C05450=1081.864,342.520,-93.492,176.172,26.985,154.564
C05451=1081.871,342.768,-93.526,176.175,26.990,154.565
C05452=1081.876,343.015,-93.561,176.178,26.994,154.566
C05453=1081.883,343.263,-93.595,176.181,27.000,154.567
C05454=1081.892,343.670,-93.651,176.186,27.008,154.568
C05455=1081.902,344.077,-93.708,176.192,27.016,154.570
C05456=1081.912,344.484,-93.765,176.197,27.024,154.571
C05457=1081.922,344.891,-93.822,176.202,27.033,154.572
C05458=1081.928,345.139,-93.856,176.205,27.038,154.573
C05459=1081.934,345.386,-93.892,176.208,27.043,154.574
C05460=1081.940,345.634,-93.926,176.212,27.048,154.575
C05461=1081.946,345.881,-93.960,176.215,27.053,154.576
C05462=1081.952,346.129,-93.996,176.218,27.058,154.577
C05463=1081.958,346.376,-94.030,176.221,27.063,154.577
C05464=1081.964,346.624,-94.066,176.224,27.068,154.578
C05465=1081.970,346.871,-94.100,176.228,27.074,154.579
C05466=1081.976,347.119,-94.135,176.231,27.078,154.580
C05467=1081.982,347.366,-94.169,176.234,27.084,154.581
C05468=1081.988,347.614,-94.204,176.237,27.088,154.582
C05469=1081.994,347.861,-94.239,176.241,27.094,154.582
C05470=1082.000,348.109,-94.274,176.244,27.099,154.583
C05471=1082.006,348.356,-94.309,176.247,27.104,154.584
C05472=1082.012,348.603,-94.344,176.251,27.110,154.585
C05473=1082.017,348.851,-94.379,176.254,27.115,154.586
C05474=1082.024,349.098,-94.414,176.256,27.120,154.587
C05475=1082.030,349.347,-94.449,176.259,27.125,154.588
C05476=1082.036,349.593,-94.484,176.263,27.130,154.589
C05477=1082.042,349.841,-94.519,176.266,27.136,154.589
C05478=1082.048,350.088,-94.553,176.269,27.141,154.590
C05479=1082.054,350.336,-94.589,176.272,27.146,154.591
C05480=1082.061,350.583,-94.624,176.276,27.152,154.592
C05481=1082.066,350.831,-94.659,176.279,27.156,154.593
C05482=1082.073,351.078,-94.694,176.282,27.162,154.594
C05483=1082.078,351.325,-94.729,176.286,27.167,154.595
C05484=1082.084,351.573,-94.765,176.289,27.172,154.596
C05485=1082.091,351.821,-94.800,176.292,27.178,154.597
C05486=1082.096,352.068,-94.835,176.296,27.183,154.598
C05487=1082.103,352.315,-94.870,176.299,27.188,154.598
C05488=1082.109,352.563,-94.906,176.302,27.194,154.599
C05489=1082.115,352.811,-94.942,176.305,27.199,154.600
C05490=1082.121,353.058,-94.976,176.308,27.204,154.601
C05491=1082.127,353.306,-95.011,176.311,27.210,154.602
C05492=1082.133,353.553,-95.047,176.315,27.215,154.603
C05493=1082.139,353.800,-95.082,176.318,27.220,154.604
C05494=1082.145,354.048,-95.118,176.321,27.226,154.605
C05495=1082.151,354.295,-95.153,176.325,27.232,154.606
C05496=1082.156,354.542,-95.189,176.328,27.237,154.607
C05497=1082.163,354.790,-95.224,176.331,27.242,154.608
C05498=1082.169,355.037,-95.260,176.335,27.248,154.609
C05499=1082.175,355.284,-95.295,176.338,27.253,154.610
C05500=1082.181,355.532,-95.331,176.340,27.258,154.611
C05501=1082.187,355.780,-95.366,176.344,27.264,154.611
C05502=1082.194,356.026,-95.402,176.347,27.270,154.612
C05503=1082.199,356.273,-95.438,176.350,27.275,154.613
C05504=1082.205,356.521,-95.473,176.354,27.280,154.614
C05505=1082.211,356.769,-95.509,176.357,27.286,154.615
C05506=1082.222,357.179,-95.568,176.362,27.295,154.617
C05507=1082.232,357.589,-95.627,176.368,27.304,154.618
C05508=1082.242,357.998,-95.687,176.374,27.313,154.620
C05509=1082.251,358.408,-95.746,176.379,27.322,154.622
C05510=1082.258,358.656,-95.781,176.383,27.328,154.623
C05511=1082.265,358.903,-95.818,176.386,27.334,154.624
C05512=1082.271,359.150,-95.853,176.388,27.339,154.625
C05513=1082.277,359.398,-95.889,176.392,27.345,154.625
C05514=1082.283,359.645,-95.925,176.395,27.351,154.626
C05515=1082.288,359.892,-95.961,176.399,27.357,154.628
C05516=1082.295,360.139,-95.997,176.402,27.362,154.628
C05517=1082.301,360.387,-96.033,176.405,27.367,154.629
C05518=1082.307,360.635,-96.069,176.409,27.373,154.630
C05519=1082.313,360.882,-96.105,176.412,27.379,154.632
C05520=1082.319,361.129,-96.141,176.416,27.385,154.632
C05521=1082.325,361.376,-96.177,176.418,27.390,154.633
C05522=1082.332,361.624,-96.213,176.421,27.396,154.635
C05523=1082.337,361.870,-96.249,176.425,27.402,154.636
C05524=1082.344,362.117,-96.286,176.428,27.408,154.637
C05525=1082.350,362.365,-96.321,176.432,27.413,154.637
C05526=1082.356,362.612,-96.358,176.435,27.419,154.639
C05527=1082.362,362.860,-96.394,176.439,27.425,154.640
C05528=1082.368,363.107,-96.431,176.442,27.431,154.641
C05529=1082.374,363.354,-96.467,176.445,27.437,154.642
C05530=1082.380,363.602,-96.503,176.448,27.442,154.643
C05531=1082.386,363.849,-96.539,176.452,27.448,154.644
C05532=1082.393,364.096,-96.576,176.455,27.454,154.645
C05533=1082.399,364.343,-96.612,176.458,27.460,154.646
C05534=1082.405,364.591,-96.648,176.462,27.466,154.647
C05535=1082.411,364.838,-96.684,176.465,27.471,154.648
C05536=1082.417,365.085,-96.721,176.468,27.477,154.649
C05537=1082.423,365.332,-96.758,176.471,27.483,154.650
C05538=1082.430,365.579,-96.794,176.475,27.489,154.651
C05539=1082.436,365.826,-96.831,176.478,27.495,154.652
C05540=1082.442,366.074,-96.868,176.482,27.501,154.653
C05541=1082.448,366.321,-96.903,176.485,27.507,154.654
C05542=1082.454,366.568,-96.940,176.489,27.513,154.655
C05543=1082.459,366.816,-96.977,176.491,27.519,154.656
C05544=1082.466,367.063,-97.013,176.495,27.525,154.658
C05545=1082.472,367.310,-97.050,176.498,27.531,154.659
C05546=1082.478,367.557,-97.087,176.502,27.538,154.660
C05547=1082.484,367.804,-97.123,176.505,27.543,154.661
C05548=1082.490,368.052,-97.160,176.509,27.550,154.662
C05549=1082.496,368.298,-97.197,176.511,27.555,154.663
C05550=1082.503,368.545,-97.234,176.515,27.562,154.664
C05551=1082.509,368.793,-97.271,176.518,27.567,154.665
C05552=1082.515,369.040,-97.308,176.522,27.574,154.666
C05553=1082.521,369.288,-97.345,176.526,27.580,154.667
C05554=1082.527,369.535,-97.381,176.529,27.586,154.669
C05555=1082.533,369.782,-97.418,176.532,27.592,154.670
C05556=1082.539,370.029,-97.455,176.535,27.598,154.671
C05557=1082.546,370.276,-97.492,176.539,27.605,154.672
C05558=1082.552,370.489,-97.524,176.542,27.610,154.673
C05559=1082.556,370.701,-97.556,176.545,27.615,154.674
C05560=1082.562,370.915,-97.588,176.547,27.620,154.675
C05561=1082.567,371.128,-97.619,176.550,27.625,154.676
C05562=1082.572,371.340,-97.651,176.553,27.631,154.677
C05563=1082.578,371.554,-97.684,176.556,27.636,154.678
C05564=1082.583,371.766,-97.715,176.559,27.642,154.679
C05565=1082.589,371.979,-97.747,176.562,27.647,154.680
C05566=1082.594,372.227,-97.784,176.566,27.653,154.681
C05567=1082.601,372.474,-97.821,176.569,27.660,154.682
C05568=1082.607,372.721,-97.859,176.572,27.666,154.683
C05569=1082.614,372.968,-97.895,176.576,27.672,154.684
C05570=1082.619,373.215,-97.933,176.579,27.679,154.685
C05571=1082.626,373.462,-97.970,176.583,27.685,154.687
C05572=1082.632,373.709,-98.008,176.586,27.691,154.688
C05573=1082.639,373.956,-98.044,176.590,27.698,154.689
C05574=1082.645,374.203,-98.082,176.593,27.704,154.690
C05575=1082.650,374.450,-98.119,176.596,27.710,154.691
C05576=1082.657,374.698,-98.156,176.600,27.717,154.692
C05577=1082.663,374.944,-98.194,176.603,27.723,154.694
C05578=1082.669,375.192,-98.231,176.607,27.730,154.695
C05579=1082.675,375.438,-98.269,176.610,27.736,154.696
C05580=1082.682,375.686,-98.307,176.613,27.743,154.697
C05581=1082.688,375.933,-98.344,176.617,27.749,154.698
C05582=1082.694,376.180,-98.381,176.621,27.756,154.700
C05583=1082.700,376.427,-98.419,176.624,27.762,154.701
C05584=1082.707,376.674,-98.457,176.627,27.769,154.702
C05585=1082.712,376.921,-98.494,176.630,27.775,154.703
C05586=1082.719,377.168,-98.532,176.634,27.782,154.705
C05587=1082.725,377.415,-98.570,176.638,27.788,154.706
C05588=1082.731,377.662,-98.607,176.640,27.795,154.707
C05589=1082.738,377.909,-98.645,176.644,27.802,154.708
C05590=1082.744,378.156,-98.683,176.648,27.808,154.710
C05591=1082.750,378.403,-98.720,176.651,27.815,154.711
C05592=1082.756,378.650,-98.758,176.655,27.821,154.712
C05593=1082.762,378.897,-98.796,176.658,27.828,154.713
C05594=1082.769,379.143,-98.833,176.661,27.835,154.715
C05595=1082.775,379.391,-98.871,176.665,27.841,154.716
C05596=1082.781,379.637,-98.909,176.669,27.848,154.717
C05597=1082.788,379.885,-98.947,176.672,27.855,154.718
C05598=1082.794,380.132,-98.985,176.675,27.862,154.720
C05599=1082.800,380.379,-99.023,176.679,27.869,154.721
C05600=1082.807,380.625,-99.060,176.683,27.875,154.722
C05601=1082.813,380.873,-99.099,176.686,27.882,154.723
C05602=1082.819,381.120,-99.136,176.689,27.888,154.725
C05603=1082.826,381.367,-99.174,176.693,27.895,154.726
C05604=1082.832,381.613,-99.213,176.697,27.902,154.727
C05605=1082.838,381.861,-99.251,176.700,27.909,154.728
C05606=1082.844,382.107,-99.289,176.704,27.916,154.730
C05607=1082.851,382.355,-99.327,176.707,27.923,154.731
C05608=1082.857,382.601,-99.365,176.711,27.930,154.732
C05609=1082.863,382.848,-99.403,176.714,27.937,154.734
C05610=1082.869,383.095,-99.441,176.718,27.943,154.735
C05611=1082.876,383.341,-99.480,176.721,27.951,154.736
C05612=1082.882,383.589,-99.518,176.725,27.958,154.738
C05613=1082.889,383.836,-99.556,176.728,27.965,154.739
C05614=1082.893,384.062,-99.592,176.732,27.971,154.740
C05615=1082.899,384.290,-99.626,176.734,27.978,154.742
C05616=1082.905,384.517,-99.662,176.737,27.984,154.743
C05617=1082.911,384.745,-99.697,176.741,27.991,154.744
C05618=1082.917,384.971,-99.733,176.744,27.997,154.745
C05619=1082.923,385.199,-99.768,176.748,28.004,154.747
C05620=1082.928,385.426,-99.804,176.751,28.010,154.748
C05621=1082.934,385.652,-99.839,176.753,28.017,154.749
C05622=1082.941,385.900,-99.877,176.757,28.024,154.751
C05623=1082.946,386.146,-99.916,176.761,28.031,154.752
C05624=1082.953,386.394,-99.954,176.765,28.038,154.753
C05625=1082.959,386.640,-99.993,176.768,28.046,154.755
C05626=1082.966,386.887,-100.032,176.772,28.053,154.756
C05627=1082.972,387.134,-100.070,176.775,28.060,154.757
C05628=1082.978,387.380,-100.109,176.779,28.067,154.759
C05629=1082.985,387.627,-100.148,176.782,28.074,154.760
C05630=1082.992,387.874,-100.187,176.786,28.082,154.762
C05631=1082.997,388.121,-100.224,176.790,28.089,154.763
C05632=1083.004,388.368,-100.264,176.794,28.096,154.764
C05633=1083.010,388.615,-100.303,176.796,28.103,154.766
C05634=1083.017,388.861,-100.341,176.800,28.111,154.767
C05635=1083.023,389.108,-100.380,176.804,28.118,154.769
C05636=1083.029,389.355,-100.419,176.807,28.126,154.770
C05637=1083.036,389.602,-100.457,176.811,28.133,154.772
C05638=1083.042,389.848,-100.496,176.815,28.140,154.773
C05639=1083.048,390.096,-100.535,176.819,28.148,154.774
C05640=1083.055,390.342,-100.574,176.822,28.155,154.776
C05641=1083.062,390.589,-100.613,176.826,28.163,154.777
C05642=1083.069,390.836,-100.652,176.829,28.170,154.779
C05643=1083.074,391.083,-100.691,176.833,28.177,154.780
C05644=1083.081,391.329,-100.730,176.836,28.185,154.782
C05645=1083.088,391.576,-100.769,176.840,28.192,154.783
C05646=1083.094,391.823,-100.809,176.844,28.200,154.785
C05647=1083.101,392.070,-100.848,176.847,28.208,154.786
C05648=1083.106,392.316,-100.887,176.851,28.215,154.788
C05649=1083.113,392.563,-100.925,176.855,28.223,154.789
C05650=1083.119,392.810,-100.965,176.858,28.231,154.791
C05651=1083.126,393.057,-101.004,176.862,28.239,154.792
C05652=1083.133,393.303,-101.044,176.866,28.246,154.794
C05653=1083.139,393.550,-101.083,176.869,28.254,154.795
C05654=1083.145,393.797,-101.122,176.872,28.261,154.797
C05655=1083.152,394.044,-101.162,176.876,28.269,154.798
C05656=1083.158,394.290,-101.201,176.880,28.277,154.800
C05657=1083.164,394.537,-101.240,176.883,28.285,154.801
C05658=1083.171,394.783,-101.280,176.887,28.292,154.803
C05659=1083.177,395.030,-101.319,176.891,28.300,154.805
C05660=1083.183,395.277,-101.359,176.894,28.308,154.806
C05661=1083.190,395.524,-101.399,176.898,28.316,154.808
C05662=1083.197,395.771,-101.438,176.902,28.324,154.809
C05663=1083.203,396.017,-101.478,176.905,28.332,154.811
C05664=1083.209,396.264,-101.517,176.909,28.340,154.812
C05665=1083.216,396.511,-101.557,176.913,28.348,154.814
C05666=1083.222,396.758,-101.596,176.916,28.356,154.816
C05667=1083.229,397.004,-101.636,176.920,28.364,154.817
C05668=1083.235,397.251,-101.676,176.924,28.372,154.819
C05669=1083.242,397.498,-101.715,176.927,28.380,154.820
C05670=1083.248,397.732,-101.753,176.931,28.388,154.822
C05671=1083.254,397.966,-101.791,176.935,28.395,154.823
C05672=1083.260,398.200,-101.829,176.938,28.403,154.825
C05673=1083.266,398.435,-101.867,176.941,28.411,154.827
C05674=1083.272,398.669,-101.905,176.945,28.418,154.828
C05675=1083.278,398.903,-101.942,176.949,28.426,154.830
C05676=1083.285,399.137,-101.980,176.953,28.434,154.831
C05677=1083.291,399.371,-102.018,176.955,28.441,154.833
C05678=1083.298,399.618,-102.058,176.959,28.450,154.834
C05679=1083.304,399.864,-102.098,176.963,28.458,154.836
C05680=1083.310,400.111,-102.138,176.967,28.467,154.838
C05681=1083.317,400.357,-102.178,176.971,28.475,154.840
C05682=1083.323,400.604,-102.219,176.974,28.483,154.841
C05683=1083.330,400.851,-102.259,176.978,28.492,154.843
C05684=1083.336,401.097,-102.299,176.982,28.500,154.845
C05685=1083.342,401.345,-102.339,176.985,28.508,154.846
C05686=1083.349,401.591,-102.379,176.989,28.517,154.848
C05687=1083.356,401.837,-102.420,176.993,28.525,154.850
C05688=1083.363,402.084,-102.460,176.996,28.534,154.851
C05689=1083.369,402.331,-102.500,177.000,28.542,154.853
C05690=1083.375,402.577,-102.540,177.005,28.551,154.855
C05691=1083.382,402.824,-102.581,177.008,28.559,154.857
C05692=1083.389,403.071,-102.621,177.012,28.568,154.858
C05693=1083.395,403.317,-102.661,177.016,28.576,154.860
C05694=1083.401,403.564,-102.701,177.019,28.585,154.862
C05695=1083.409,403.811,-102.743,177.023,28.593,154.864
C05696=1083.414,404.057,-102.783,177.027,28.602,154.865
C05697=1083.421,404.304,-102.824,177.031,28.611,154.867
C05698=1083.428,404.551,-102.864,177.035,28.620,154.869
C05699=1083.434,404.797,-102.905,177.038,28.628,154.871
C05700=1083.441,405.044,-102.945,177.042,28.637,154.873
C05701=1083.448,405.291,-102.986,177.047,28.646,154.874
C05702=1083.454,405.537,-103.027,177.050,28.655,154.876
C05703=1083.460,405.783,-103.067,177.054,28.663,154.878
C05704=1083.467,406.030,-103.108,177.058,28.672,154.880
C05705=1083.474,406.277,-103.149,177.061,28.681,154.882
C05706=1083.479,406.523,-103.189,177.066,28.690,154.883
C05707=1083.487,406.770,-103.231,177.069,28.699,154.885
C05708=1083.493,407.016,-103.271,177.073,28.708,154.887
C05709=1083.500,407.263,-103.312,177.077,28.717,154.889
C05710=1083.506,407.509,-103.353,177.081,28.726,154.891
C05711=1083.513,407.756,-103.394,177.085,28.735,154.893
C05712=1083.519,408.003,-103.435,177.088,28.744,154.895
C05713=1083.526,408.249,-103.476,177.093,28.753,154.897
C05714=1083.533,408.496,-103.517,177.097,28.762,154.898
C05715=1083.539,408.742,-103.558,177.100,28.772,154.900
C05716=1083.546,408.989,-103.599,177.104,28.781,154.902
C05717=1083.552,409.235,-103.641,177.108,28.790,154.904
C05718=1083.559,409.482,-103.681,177.112,28.799,154.906
C05719=1083.565,409.728,-103.723,177.116,28.808,154.908
C05720=1083.572,409.975,-103.764,177.120,28.818,154.910
C05721=1083.578,410.221,-103.806,177.124,28.827,154.912
C05722=1083.586,410.468,-103.847,177.128,28.837,154.914
C05723=1083.591,410.714,-103.888,177.132,28.846,154.916
C05724=1083.599,410.960,-103.929,177.136,28.855,154.918
C05725=1083.605,411.207,-103.971,177.140,28.865,154.920
C05726=1083.611,411.442,-104.010,177.144,28.874,154.922
C05727=1083.618,411.678,-104.050,177.148,28.883,154.924
C05728=1083.624,411.912,-104.089,177.151,28.892,154.925
C05729=1083.631,412.147,-104.129,177.155,28.901,154.927
C05730=1083.636,412.382,-104.168,177.159,28.910,154.929
C05731=1083.643,412.617,-104.208,177.163,28.919,154.931
C05732=1083.650,412.853,-104.248,177.167,28.929,154.933
C05733=1083.656,413.087,-104.287,177.171,28.938,154.935
C05734=1083.663,413.334,-104.328,177.175,28.948,154.937
C05735=1083.670,413.581,-104.370,177.179,28.957,154.939
C05736=1083.676,413.826,-104.412,177.182,28.966,154.941
C05737=1083.683,414.073,-104.454,177.187,28.976,154.943
C05738=1083.690,414.320,-104.495,177.191,28.986,154.945
C05739=1083.697,414.566,-104.537,177.195,28.996,154.947
C05740=1083.703,414.812,-104.579,177.199,29.006,154.949
C05741=1083.710,415.059,-104.621,177.203,29.015,154.951
C05742=1083.717,415.305,-104.663,177.207,29.025,154.953
C05743=1083.724,415.552,-104.704,177.211,29.035,154.956
C05744=1083.731,415.799,-104.746,177.216,29.045,154.958
C05745=1083.738,416.044,-104.788,177.220,29.055,154.960
C05746=1083.744,416.291,-104.830,177.224,29.065,154.962
C05747=1083.751,416.537,-104.872,177.228,29.075,154.964
C05748=1083.758,416.783,-104.915,177.232,29.085,154.966
C05749=1083.764,417.030,-104.956,177.236,29.095,154.968
C05750=1083.771,417.276,-104.999,177.241,29.106,154.971
C05751=1083.777,417.522,-105.041,177.245,29.116,154.973
C05752=1083.784,417.769,-105.083,177.249,29.126,154.975
C05753=1083.792,418.015,-105.125,177.253,29.136,154.977
C05754=1083.798,418.261,-105.168,177.257,29.146,154.979
C05755=1083.805,418.508,-105.210,177.261,29.157,154.982
C05756=1083.811,418.754,-105.252,177.266,29.167,154.984
C05757=1083.818,419.000,-105.294,177.270,29.177,154.986
C05758=1083.825,419.246,-105.337,177.274,29.188,154.988
C05759=1083.832,419.493,-105.379,177.279,29.198,154.990
C05760=1083.839,419.739,-105.422,177.282,29.209,154.993
C05761=1083.846,419.985,-105.464,177.287,29.219,154.995
C05762=1083.852,420.231,-105.507,177.291,29.230,154.997
C05763=1083.859,420.478,-105.549,177.295,29.240,154.999
C05764=1083.866,420.724,-105.592,177.300,29.251,155.002
C05765=1083.873,420.970,-105.634,177.304,29.261,155.004
C05766=1083.880,421.217,-105.677,177.309,29.272,155.006
C05767=1083.887,421.463,-105.719,177.312,29.283,155.008
C05768=1083.894,421.709,-105.762,177.317,29.293,155.011
C05769=1083.900,421.955,-105.805,177.321,29.304,155.013
C05770=1083.908,422.201,-105.848,177.326,29.315,155.015
C05771=1083.914,422.447,-105.890,177.330,29.326,155.018
C05772=1083.921,422.694,-105.933,177.334,29.337,155.020
C05773=1083.928,422.940,-105.977,177.339,29.348,155.022
C05774=1083.935,423.186,-106.019,177.343,29.359,155.025
C05775=1083.941,423.432,-106.062,177.347,29.369,155.027
C05776=1083.949,423.678,-106.105,177.351,29.381,155.030
C05777=1083.955,423.924,-106.148,177.356,29.392,155.032
C05778=1083.962,424.171,-106.192,177.360,29.403,155.034
C05779=1083.969,424.417,-106.234,177.365,29.414,155.037
C05780=1083.976,424.663,-106.278,177.370,29.425,155.039
C05781=1083.983,424.909,-106.321,177.373,29.436,155.042
C05782=1083.990,425.153,-106.363,177.378,29.447,155.044
C05783=1083.996,425.395,-106.406,177.382,29.459,155.047
C05784=1084.003,425.638,-106.449,177.387,29.470,155.049
C05785=1084.010,425.881,-106.492,177.391,29.481,155.051
C05786=1084.017,426.125,-106.534,177.395,29.492,155.054
C05787=1084.024,426.367,-106.577,177.400,29.503,155.056
C05788=1084.031,426.610,-106.619,177.404,29.514,155.059
C05789=1084.038,426.853,-106.663,177.409,29.526,155.061
C05790=1084.045,427.099,-106.706,177.413,29.537,155.064
C05791=1084.052,427.346,-106.749,177.418,29.549,155.066
C05792=1084.059,427.592,-106.793,177.423,29.560,155.069
C05793=1084.066,427.838,-106.836,177.427,29.572,155.071
C05794=1084.073,428.083,-106.880,177.432,29.583,155.074
C05795=1084.081,428.330,-106.923,177.436,29.595,155.076
C05796=1084.087,428.576,-106.967,177.441,29.607,155.079
C05797=1084.094,428.821,-107.010,177.445,29.619,155.082
C05798=1084.101,429.068,-107.055,177.450,29.630,155.084
C05799=1084.108,429.314,-107.098,177.454,29.642,155.087
C05800=1084.115,429.560,-107.142,177.459,29.654,155.089
C05801=1084.122,429.806,-107.187,177.464,29.666,155.092
C05802=1084.129,430.051,-107.230,177.468,29.678,155.095
C05803=1084.136,430.297,-107.274,177.473,29.690,155.097
C05804=1084.143,430.544,-107.317,177.477,29.702,155.100
C05805=1084.150,430.789,-107.362,177.482,29.714,155.103
C05806=1084.158,431.035,-107.406,177.486,29.726,155.105
C05807=1084.164,431.281,-107.449,177.491,29.738,155.108
C05808=1084.172,431.527,-107.494,177.496,29.751,155.111
C05809=1084.179,431.773,-107.538,177.500,29.763,155.114
C05810=1084.186,432.019,-107.583,177.505,29.775,155.116
C05811=1084.193,432.265,-107.626,177.510,29.787,155.119
C05812=1084.200,432.511,-107.670,177.515,29.800,155.122
C05813=1084.207,432.757,-107.715,177.520,29.812,155.124
C05814=1084.214,433.003,-107.760,177.524,29.825,155.127
C05815=1084.221,433.249,-107.803,177.529,29.837,155.130
C05816=1084.228,433.495,-107.848,177.533,29.850,155.133
C05817=1084.236,433.740,-107.892,177.538,29.862,155.136
C05818=1084.243,433.987,-107.936,177.543,29.875,155.138
C05819=1084.249,434.232,-107.981,177.548,29.888,155.141
C05820=1084.257,434.478,-108.026,177.553,29.900,155.144
C05821=1084.263,434.723,-108.071,177.557,29.913,155.147
C05822=1084.271,434.969,-108.115,177.562,29.926,155.150
C05823=1084.278,435.216,-108.160,177.567,29.939,155.153
C05824=1084.285,435.461,-108.204,177.572,29.951,155.156
C05825=1084.293,435.707,-108.249,177.577,29.964,155.159
C05826=1084.299,435.953,-108.293,177.581,29.977,155.162
C05827=1084.307,436.199,-108.338,177.587,29.991,155.164
C05828=1084.314,436.444,-108.384,177.591,30.003,155.167
C05829=1084.322,436.690,-108.429,177.596,30.016,155.170
C05830=1084.328,436.935,-108.473,177.601,30.030,155.173
C05831=1084.336,437.182,-108.518,177.606,30.043,155.176
C05832=1084.343,437.428,-108.563,177.611,30.056,155.179
C05833=1084.350,437.674,-108.608,177.616,30.070,155.182
C05834=1084.357,437.918,-108.653,177.621,30.083,155.185
C05835=1084.365,438.164,-108.698,177.626,30.096,155.188
C05836=1084.372,438.410,-108.743,177.631,30.110,155.191
C05837=1084.380,438.656,-108.789,177.636,30.123,155.194
C05838=1084.390,439.030,-108.857,177.644,30.143,155.199
C05839=1084.401,439.404,-108.926,177.652,30.164,155.204
C05840=1084.413,439.779,-108.995,177.658,30.185,155.209
C05841=1084.424,440.153,-109.064,177.666,30.206,155.213
C05842=1084.431,440.399,-109.110,177.672,30.220,155.216
C05843=1084.439,440.644,-109.155,177.677,30.234,155.220
C05844=1084.446,440.890,-109.200,177.682,30.247,155.223
C05845=1084.453,441.136,-109.247,177.687,30.261,155.226
C05846=1084.461,441.381,-109.292,177.693,30.276,155.229
C05847=1084.468,441.627,-109.338,177.697,30.290,155.232
C05848=1084.476,441.873,-109.383,177.703,30.304,155.236
C05849=1084.483,442.118,-109.429,177.707,30.318,155.239
C05850=1084.490,442.364,-109.475,177.713,30.332,155.242
C05851=1084.498,442.609,-109.520,177.718,30.346,155.245
C05852=1084.505,442.855,-109.567,177.723,30.361,155.249
C05853=1084.513,443.101,-109.612,177.728,30.375,155.252
C05854=1084.520,443.346,-109.658,177.734,30.389,155.255
C05855=1084.527,443.592,-109.704,177.739,30.404,155.259
C05856=1084.535,443.837,-109.750,177.744,30.418,155.262
C05857=1084.542,444.082,-109.797,177.750,30.433,155.265
C05858=1084.550,444.328,-109.842,177.754,30.447,155.269
C05859=1084.557,444.573,-109.888,177.760,30.462,155.272
C05860=1084.565,444.820,-109.935,177.766,30.477,155.275
C05861=1084.573,445.064,-109.981,177.770,30.492,155.279
C05862=1084.580,445.310,-110.027,177.776,30.507,155.282
C05863=1084.587,445.556,-110.073,177.781,30.521,155.286
C05864=1084.594,445.801,-110.120,177.787,30.536,155.289
C05865=1084.602,446.046,-110.166,177.790,30.551,155.293
C05866=1084.610,446.292,-110.213,177.795,30.566,155.296
C05867=1084.617,446.538,-110.259,177.799,30.580,155.300
C05868=1084.625,446.782,-110.305,177.804,30.595,155.303
C05869=1084.632,447.028,-110.352,177.807,30.610,155.307
C05870=1084.640,447.274,-110.398,177.810,30.625,155.310
C05871=1084.647,447.519,-110.445,177.814,30.639,155.314
C05872=1084.654,447.765,-110.492,177.817,30.654,155.317
C05873=1084.663,448.010,-110.538,177.820,30.669,155.321
C05874=1084.670,448.255,-110.585,177.822,30.683,155.325
C05875=1084.678,448.500,-110.632,177.825,30.698,155.328
C05876=1084.685,448.746,-110.678,177.827,30.713,155.332
C05877=1084.693,448.992,-110.725,177.830,30.727,155.335
C05878=1084.701,449.236,-110.772,177.832,30.742,155.339
C05879=1084.709,449.481,-110.819,177.834,30.757,155.343
C05880=1084.718,449.727,-110.864,177.836,30.770,155.346
C05881=1084.730,449.973,-110.908,177.838,30.783,155.349
C05882=1084.358,449.965,-111.117,177.805,30.963,155.398
C05883=1084.345,449.719,-111.072,177.802,30.951,155.395
C05884=1084.336,449.474,-111.026,177.800,30.937,155.391
C05885=1084.327,449.228,-110.980,177.798,30.923,155.388
C05886=1084.320,448.984,-110.934,177.796,30.908,155.384
C05887=1084.313,448.767,-110.892,177.794,30.895,155.381
C05888=1084.306,448.551,-110.850,177.792,30.882,155.378
C05889=1084.299,448.334,-110.809,177.789,30.869,155.374
C05890=1084.292,448.117,-110.768,177.787,30.856,155.371
C05891=1084.286,447.900,-110.727,177.784,30.843,155.368
C05892=1084.279,447.683,-110.685,177.782,30.830,155.365
C05893=1084.272,447.466,-110.644,177.779,30.817,155.362
C05894=1084.265,447.249,-110.603,177.776,30.804,155.358
C05895=1084.258,447.004,-110.556,177.772,30.789,155.355
C05896=1084.251,446.759,-110.510,177.768,30.775,155.351
C05897=1084.243,446.513,-110.463,177.764,30.760,155.348
C05898=1084.235,446.268,-110.416,177.759,30.745,155.344
C05899=1084.228,446.023,-110.370,177.756,30.730,155.341
C05900=1084.220,445.777,-110.323,177.751,30.715,155.337
C05901=1084.213,445.531,-110.277,177.745,30.700,155.334
C05902=1084.205,445.286,-110.230,177.740,30.686,155.330
C05903=1084.198,445.040,-110.184,177.734,30.671,155.327
C05904=1084.190,444.796,-110.138,177.729,30.656,155.324
C05905=1084.183,444.549,-110.091,177.724,30.641,155.320
C05906=1084.175,444.304,-110.045,177.718,30.627,155.317
C05907=1084.167,444.058,-110.000,177.713,30.612,155.313
C05908=1084.160,443.813,-109.953,177.707,30.597,155.310
C05909=1084.153,443.568,-109.907,177.703,30.583,155.307
C05910=1084.146,443.322,-109.861,177.697,30.568,155.303
C05911=1084.138,443.077,-109.815,177.691,30.554,155.300
C05912=1084.130,442.831,-109.770,177.686,30.539,155.297
C05913=1084.123,442.585,-109.723,177.681,30.525,155.293
C05914=1084.116,442.340,-109.678,177.676,30.511,155.290
C05915=1084.108,442.095,-109.632,177.670,30.497,155.287
C05916=1084.101,441.849,-109.586,177.665,30.482,155.283
C05917=1084.093,441.603,-109.540,177.660,30.468,155.280
C05918=1084.086,441.358,-109.495,177.655,30.454,155.277
C05919=1084.078,441.112,-109.449,177.649,30.440,155.274
C05920=1084.071,440.867,-109.403,177.644,30.426,155.271
C05921=1084.064,440.621,-109.357,177.639,30.412,155.267
C05922=1084.057,440.375,-109.312,177.634,30.399,155.264
C05923=1084.050,440.166,-109.273,177.629,30.387,155.262
C05924=1084.043,439.958,-109.234,177.625,30.375,155.259
C05925=1084.038,439.750,-109.195,177.620,30.363,155.256
C05926=1084.032,439.541,-109.157,177.616,30.352,155.254
C05927=1084.026,439.333,-109.119,177.612,30.340,155.251
C05928=1084.019,439.125,-109.080,177.607,30.329,155.248
C05929=1084.012,438.918,-109.042,177.604,30.317,155.246
C05930=1084.006,438.709,-109.004,177.599,30.306,155.243
C05931=1083.999,438.463,-108.959,177.594,30.292,155.240
C05932=1083.991,438.217,-108.914,177.588,30.279,155.237
C05933=1083.984,437.971,-108.869,177.584,30.265,155.234
C05934=1083.976,437.726,-108.823,177.579,30.252,155.231
C05935=1083.969,437.480,-108.778,177.573,30.239,155.228
C05936=1083.962,437.235,-108.734,177.568,30.226,155.225
C05937=1083.955,436.989,-108.688,177.564,30.212,155.222
C05938=1083.947,436.743,-108.643,177.559,30.199,155.219
C05939=1083.940,436.497,-108.598,177.553,30.186,155.216
C05940=1083.933,436.252,-108.554,177.549,30.173,155.213
C05941=1083.926,436.006,-108.509,177.544,30.160,155.210
C05942=1083.919,435.760,-108.464,177.538,30.147,155.207
C05943=1083.912,435.514,-108.419,177.534,30.134,155.204
C05944=1083.904,435.268,-108.374,177.529,30.121,155.201
C05945=1083.897,435.022,-108.329,177.524,30.108,155.199
C05946=1083.890,434.777,-108.285,177.519,30.095,155.196
C05947=1083.883,434.531,-108.240,177.514,30.083,155.193
C05948=1083.875,434.285,-108.195,177.509,30.070,155.190
C05949=1083.868,434.040,-108.151,177.505,30.057,155.187
C05950=1083.861,433.793,-108.106,177.500,30.045,155.184
C05951=1083.855,433.548,-108.062,177.495,30.032,155.181
C05952=1083.847,433.301,-108.017,177.490,30.019,155.179
C05953=1083.840,433.056,-107.973,177.485,30.007,155.176
C05954=1083.833,432.810,-107.928,177.480,29.994,155.173
C05955=1083.826,432.564,-107.884,177.476,29.982,155.170
C05956=1083.819,432.318,-107.840,177.471,29.970,155.167
C05957=1083.812,432.072,-107.795,177.466,29.957,155.165
C05958=1083.804,431.827,-107.751,177.462,29.945,155.162
C05959=1083.797,431.580,-107.707,177.457,29.932,155.159
C05960=1083.790,431.335,-107.663,177.451,29.920,155.157
C05961=1083.783,431.088,-107.619,177.447,29.908,155.154
C05962=1083.776,430.843,-107.574,177.442,29.896,155.151
C05963=1083.769,430.597,-107.531,177.437,29.884,155.148
C05964=1083.762,430.351,-107.487,177.433,29.872,155.146
C05965=1083.755,430.105,-107.442,177.428,29.860,155.143
C05966=1083.747,429.859,-107.399,177.423,29.848,155.140
C05967=1083.741,429.613,-107.355,177.419,29.836,155.138
C05968=1083.733,429.366,-107.311,177.414,29.824,155.135
C05969=1083.726,429.121,-107.267,177.409,29.812,155.133
C05970=1083.720,428.875,-107.223,177.405,29.800,155.130
C05971=1083.712,428.629,-107.179,177.400,29.788,155.127
C05972=1083.706,428.383,-107.135,177.395,29.777,155.125
C05973=1083.698,428.137,-107.092,177.391,29.765,155.122
C05974=1083.691,427.891,-107.048,177.386,29.753,155.120
C05975=1083.684,427.645,-107.005,177.382,29.742,155.117
C05976=1083.677,427.399,-106.961,177.377,29.730,155.114
C05977=1083.669,427.153,-106.918,177.372,29.718,155.112
C05978=1083.663,426.907,-106.874,177.368,29.707,155.109
C05979=1083.656,426.664,-106.831,177.364,29.696,155.107
C05980=1083.649,426.419,-106.788,177.359,29.685,155.104
C05981=1083.642,426.176,-106.745,177.355,29.673,155.102
C05982=1083.635,425.933,-106.702,177.350,29.662,155.100
C05983=1083.628,425.688,-106.659,177.345,29.651,155.097
C05984=1083.621,425.444,-106.617,177.341,29.640,155.095
C05985=1083.614,425.201,-106.574,177.337,29.629,155.092
C05986=1083.608,424.957,-106.531,177.332,29.617,155.090
C05987=1083.600,424.711,-106.487,177.328,29.606,155.087
C05988=1083.594,424.465,-106.445,177.323,29.595,155.085
C05989=1083.586,424.219,-106.402,177.318,29.584,155.082
C05990=1083.580,423.973,-106.358,177.315,29.573,155.080
C05991=1083.573,423.727,-106.315,177.310,29.561,155.078
C05992=1083.566,423.481,-106.273,177.306,29.551,155.075
C05993=1083.559,423.235,-106.229,177.301,29.540,155.073
C05994=1083.553,422.988,-106.186,177.296,29.528,155.070
C05995=1083.545,422.742,-106.143,177.293,29.517,155.068
C05996=1083.538,422.496,-106.100,177.288,29.507,155.066
C05997=1083.532,422.249,-106.058,177.283,29.496,155.063
C05998=1083.524,422.004,-106.014,177.279,29.485,155.061
C05999=1083.518,421.757,-105.972,177.275,29.474,155.059
C06000=1083.511,421.511,-105.929,177.270,29.464,155.056
C06001=1083.505,421.265,-105.886,177.266,29.453,155.054
C06002=1083.498,421.018,-105.844,177.261,29.442,155.052
C06003=1083.491,420.772,-105.801,177.258,29.432,155.050
C06004=1083.484,420.526,-105.758,177.253,29.421,155.047
C06005=1083.476,420.280,-105.716,177.248,29.410,155.045
C06006=1083.469,420.034,-105.673,177.245,29.400,155.043
C06007=1083.462,419.788,-105.631,177.240,29.390,155.040
C06008=1083.455,419.542,-105.588,177.235,29.379,155.038
C06009=1083.449,419.295,-105.546,177.232,29.368,155.036
C06010=1083.442,419.049,-105.503,177.227,29.358,155.034
C06011=1083.435,418.802,-105.461,177.222,29.347,155.031
C06012=1083.428,418.556,-105.419,177.219,29.337,155.029
C06013=1083.422,418.310,-105.376,177.214,29.327,155.027
C06014=1083.415,418.064,-105.334,177.210,29.317,155.025
C06015=1083.408,417.818,-105.291,177.206,29.306,155.023
C06016=1083.402,417.571,-105.249,177.201,29.296,155.020
C06017=1083.395,417.324,-105.207,177.198,29.286,155.018
C06018=1083.388,417.078,-105.165,177.193,29.276,155.016
C06019=1083.381,416.832,-105.122,177.189,29.266,155.014
C06020=1083.374,416.585,-105.081,177.185,29.255,155.012
C06021=1083.368,416.340,-105.039,177.180,29.245,155.010
C06022=1083.361,416.093,-104.996,177.176,29.235,155.007
C06023=1083.354,415.847,-104.954,177.172,29.225,155.005
C06024=1083.347,415.600,-104.912,177.168,29.215,155.003
C06025=1083.340,415.354,-104.870,177.163,29.205,155.001
C06026=1083.334,415.108,-104.828,177.160,29.195,154.999
C06027=1083.327,414.861,-104.786,177.155,29.185,154.997
C06028=1083.320,414.615,-104.745,177.151,29.176,154.995
C06029=1083.313,414.368,-104.703,177.147,29.166,154.993
C06030=1083.306,414.122,-104.661,177.143,29.156,154.991
C06031=1083.300,413.875,-104.620,177.139,29.146,154.989
C06032=1083.293,413.629,-104.577,177.135,29.137,154.987
C06033=1083.286,413.383,-104.536,177.130,29.127,154.985
C06034=1083.279,413.136,-104.494,177.127,29.117,154.983
C06035=1083.273,412.901,-104.455,177.123,29.108,154.981
C06036=1083.266,412.665,-104.415,177.119,29.099,154.979
C06037=1083.260,412.429,-104.375,177.114,29.090,154.977
C06038=1083.254,412.194,-104.335,177.111,29.081,154.975
C06039=1083.247,411.958,-104.296,177.107,29.071,154.973
C06040=1083.241,411.723,-104.256,177.103,29.062,154.971
C06041=1083.234,411.486,-104.216,177.100,29.053,154.969
C06042=1083.228,411.251,-104.177,177.096,29.044,154.967
C06043=1083.222,411.004,-104.136,177.091,29.035,154.965
C06044=1083.215,410.758,-104.094,177.087,29.026,154.963
C06045=1083.209,410.512,-104.053,177.084,29.016,154.961
C06046=1083.201,410.265,-104.012,177.079,29.007,154.959
C06047=1083.195,410.018,-103.970,177.075,28.998,154.957
C06048=1083.188,409.772,-103.929,177.072,28.988,154.955
C06049=1083.182,409.525,-103.887,177.067,28.979,154.953
C06050=1083.175,409.279,-103.846,177.064,28.969,154.952
C06051=1083.168,409.032,-103.804,177.060,28.960,154.950
C06052=1083.162,408.787,-103.764,177.055,28.951,154.948
C06053=1083.155,408.539,-103.723,177.052,28.942,154.946
C06054=1083.149,408.293,-103.682,177.048,28.933,154.944
C06055=1083.141,408.046,-103.640,177.043,28.923,154.942
C06056=1083.136,407.800,-103.599,177.040,28.914,154.940
C06057=1083.129,407.554,-103.559,177.036,28.905,154.938
C06058=1083.123,407.307,-103.517,177.032,28.896,154.936
C06059=1083.116,407.060,-103.477,177.028,28.887,154.934
C06060=1083.109,406.814,-103.436,177.024,28.878,154.933
C06061=1083.102,406.568,-103.395,177.020,28.869,154.931
C06062=1083.096,406.320,-103.354,177.016,28.860,154.929
C06063=1083.089,406.074,-103.313,177.012,28.851,154.927
C06064=1083.083,405.828,-103.273,177.008,28.842,154.925
C06065=1083.076,405.581,-103.231,177.004,28.834,154.923
C06066=1083.070,405.335,-103.191,177.001,28.825,154.922
C06067=1083.063,405.087,-103.150,176.997,28.816,154.920
C06068=1083.056,404.841,-103.109,176.992,28.807,154.918
C06069=1083.050,404.595,-103.069,176.989,28.798,154.916
C06070=1083.043,404.348,-103.029,176.985,28.790,154.914
C06071=1083.037,404.101,-102.987,176.981,28.781,154.913
C06072=1083.031,403.855,-102.947,176.978,28.772,154.911
C06073=1083.024,403.608,-102.906,176.974,28.764,154.909
C06074=1083.017,403.362,-102.866,176.969,28.755,154.907
C06075=1083.011,403.115,-102.825,176.966,28.746,154.906
C06076=1083.004,402.868,-102.785,176.962,28.738,154.904
C06077=1082.997,402.622,-102.745,176.958,28.729,154.902
C06078=1082.991,402.375,-102.705,176.955,28.721,154.900
C06079=1082.984,402.129,-102.664,176.951,28.712,154.899
C06080=1082.977,401.881,-102.624,176.947,28.704,154.897
C06081=1082.971,401.635,-102.583,176.943,28.695,154.895
C06082=1082.964,401.389,-102.543,176.939,28.687,154.893
C06083=1082.958,401.142,-102.503,176.935,28.679,154.892
C06084=1082.952,400.896,-102.463,176.931,28.670,154.890
C06085=1082.945,400.649,-102.422,176.928,28.662,154.888
C06086=1082.938,400.402,-102.382,176.924,28.653,154.887
C06087=1082.932,400.155,-102.343,176.920,28.645,154.885
C06088=1082.926,399.909,-102.302,176.917,28.636,154.883
C06089=1082.919,399.662,-102.262,176.913,28.628,154.881
C06090=1082.913,399.416,-102.222,176.909,28.620,154.880
C06091=1082.907,399.181,-102.184,176.905,28.612,154.878
C06092=1082.900,398.946,-102.146,176.902,28.604,154.877
C06093=1082.893,398.711,-102.108,176.899,28.597,154.875
C06094=1082.889,398.476,-102.070,176.895,28.589,154.874
C06095=1082.882,398.241,-102.032,176.891,28.581,154.872
C06096=1082.876,398.007,-101.994,176.887,28.573,154.870
C06097=1082.870,397.773,-101.956,176.884,28.566,154.869
C06098=1082.863,397.537,-101.918,176.881,28.558,154.867
C06099=1082.857,397.291,-101.878,176.877,28.550,154.866
C06100=1082.850,397.045,-101.839,176.873,28.542,154.864
C06101=1082.844,396.797,-101.799,176.870,28.534,154.862
C06102=1082.837,396.551,-101.759,176.866,28.526,154.861
C06103=1082.831,396.304,-101.720,176.862,28.518,154.859
C06104=1082.824,396.058,-101.680,176.859,28.510,154.858
C06105=1082.818,395.810,-101.641,176.855,28.502,154.856
C06106=1082.812,395.564,-101.601,176.851,28.494,154.855
C06107=1082.806,395.317,-101.561,176.847,28.486,154.853
C06108=1082.799,395.071,-101.522,176.844,28.478,154.851
C06109=1082.793,394.823,-101.482,176.840,28.470,154.850
C06110=1082.786,394.577,-101.442,176.836,28.463,154.848
C06111=1082.779,394.330,-101.403,176.832,28.455,154.847
C06112=1082.773,394.083,-101.364,176.829,28.447,154.845
C06113=1082.766,393.837,-101.324,176.825,28.439,154.844
C06114=1082.760,393.590,-101.285,176.821,28.431,154.842
C06115=1082.753,393.343,-101.246,176.817,28.424,154.841
C06116=1082.747,393.096,-101.206,176.814,28.416,154.839
C06117=1082.741,392.850,-101.167,176.811,28.408,154.837
C06118=1082.735,392.603,-101.128,176.807,28.401,154.836
C06119=1082.729,392.356,-101.088,176.804,28.393,154.834
C06120=1082.721,392.110,-101.049,176.800,28.385,154.833
C06121=1082.715,391.863,-101.009,176.796,28.378,154.831
C06122=1082.709,391.616,-100.971,176.792,28.370,154.830
C06123=1082.702,391.369,-100.932,176.788,28.363,154.828
C06124=1082.696,391.122,-100.893,176.785,28.355,154.827
C06125=1082.689,390.876,-100.854,176.781,28.348,154.826
C06126=1082.683,390.629,-100.815,176.777,28.340,154.824
C06127=1082.677,390.382,-100.776,176.774,28.333,154.823
C06128=1082.670,390.135,-100.737,176.771,28.325,154.821
C06129=1082.663,389.889,-100.698,176.767,28.318,154.820
C06130=1082.657,389.642,-100.659,176.763,28.310,154.818
C06131=1082.651,389.395,-100.620,176.759,28.303,154.817
C06132=1082.644,389.148,-100.581,176.756,28.295,154.815
C06133=1082.638,388.902,-100.543,176.752,28.288,154.814
C06134=1082.632,388.655,-100.503,176.748,28.281,154.812
C06135=1082.625,388.408,-100.464,176.745,28.274,154.811
C06136=1082.618,388.161,-100.426,176.742,28.266,154.810
C06137=1082.613,387.914,-100.387,176.738,28.259,154.808
C06138=1082.606,387.667,-100.348,176.734,28.252,154.807
C06139=1082.599,387.420,-100.310,176.730,28.244,154.805
C06140=1082.593,387.174,-100.271,176.727,28.237,154.804
C06141=1082.586,386.927,-100.233,176.724,28.230,154.803
C06142=1082.580,386.680,-100.194,176.720,28.223,154.801
C06143=1082.574,386.434,-100.155,176.716,28.215,154.800
C06144=1082.567,386.187,-100.116,176.712,28.208,154.798
C06145=1082.561,385.939,-100.078,176.709,28.201,154.797
C06146=1082.555,385.693,-100.040,176.706,28.194,154.796
C06147=1082.549,385.465,-100.004,176.702,28.187,154.794
C06148=1082.544,385.237,-99.969,176.699,28.181,154.793
C06149=1082.538,385.010,-99.932,176.695,28.174,154.792
C06150=1082.531,384.782,-99.897,176.692,28.168,154.791
C06151=1082.526,384.554,-99.862,176.689,28.161,154.789
C06152=1082.520,384.326,-99.827,176.686,28.154,154.788
C06153=1082.514,384.099,-99.791,176.683,28.148,154.787
C06154=1082.509,383.872,-99.756,176.679,28.141,154.786
C06155=1082.502,383.624,-99.718,176.676,28.134,154.784
C06156=1082.495,383.377,-99.679,176.672,28.127,154.783
C06157=1082.490,383.130,-99.641,176.668,28.120,154.781
C06158=1082.484,382.884,-99.602,176.666,28.114,154.780
C06159=1082.478,382.637,-99.564,176.662,28.106,154.779
C06160=1082.471,382.389,-99.526,176.658,28.099,154.777
C06161=1082.465,382.143,-99.487,176.654,28.092,154.776
C06162=1082.458,381.896,-99.449,176.651,28.086,154.775
C06163=1082.452,381.649,-99.412,176.648,28.079,154.774
C06164=1082.446,381.401,-99.373,176.644,28.072,154.772
C06165=1082.440,381.155,-99.335,176.640,28.065,154.771
C06166=1082.432,380.908,-99.298,176.637,28.058,154.770
C06167=1082.427,380.661,-99.260,176.633,28.051,154.768
C06168=1082.420,380.414,-99.222,176.630,28.044,154.767
C06169=1082.414,380.167,-99.184,176.627,28.038,154.766
C06170=1082.408,379.921,-99.146,176.623,28.031,154.765
C06171=1082.402,379.673,-99.108,176.619,28.025,154.763
C06172=1082.396,379.426,-99.070,176.616,28.018,154.762
C06173=1082.389,379.179,-99.033,176.613,28.011,154.761
C06174=1082.383,378.932,-98.995,176.609,28.004,154.759
C06175=1082.376,378.685,-98.957,176.606,27.998,154.758
C06176=1082.370,378.438,-98.919,176.602,27.991,154.757
C06177=1082.364,378.192,-98.881,176.598,27.984,154.756
C06178=1082.358,377.944,-98.843,176.595,27.978,154.754
C06179=1082.351,377.698,-98.806,176.592,27.971,154.753
C06180=1082.345,377.450,-98.768,176.588,27.965,154.752
C06181=1082.339,377.203,-98.730,176.585,27.958,154.751
C06182=1082.333,376.957,-98.692,176.581,27.952,154.750
C06183=1082.326,376.709,-98.654,176.577,27.945,154.748
C06184=1082.320,376.462,-98.618,176.574,27.939,154.747
C06185=1082.314,376.215,-98.580,176.571,27.932,154.746
C06186=1082.308,375.968,-98.542,176.568,27.925,154.745
C06187=1082.302,375.721,-98.504,176.564,27.919,154.743
C06188=1082.295,375.475,-98.467,176.560,27.912,154.742
C06189=1082.289,375.227,-98.430,176.557,27.906,154.741
C06190=1082.283,374.980,-98.392,176.553,27.899,154.740
C06191=1082.277,374.733,-98.354,176.550,27.892,154.738
C06192=1082.271,374.486,-98.318,176.547,27.886,154.737
C06193=1082.265,374.239,-98.280,176.543,27.880,154.736
C06194=1082.259,373.991,-98.243,176.540,27.874,154.735
C06195=1082.252,373.745,-98.205,176.536,27.867,154.734
C06196=1082.246,373.498,-98.168,176.533,27.861,154.732
C06197=1082.239,373.250,-98.131,176.530,27.854,154.731
C06198=1082.233,373.004,-98.093,176.526,27.848,154.730
C06199=1082.227,372.757,-98.057,176.523,27.842,154.729
C06200=1082.221,372.510,-98.019,176.519,27.835,154.728
C06201=1082.214,372.262,-97.982,176.516,27.829,154.727
C06202=1082.208,372.015,-97.945,176.512,27.823,154.726
C06203=1082.203,371.802,-97.913,176.509,27.817,154.725
C06204=1082.197,371.588,-97.880,176.506,27.812,154.724
C06205=1082.192,371.374,-97.849,176.503,27.807,154.723
C06206=1082.187,371.161,-97.816,176.500,27.801,154.722
C06207=1082.181,370.947,-97.785,176.497,27.796,154.721
C06208=1082.176,370.734,-97.753,176.494,27.790,154.720
C06209=1082.171,370.521,-97.721,176.492,27.785,154.719
C06210=1082.166,370.307,-97.689,176.489,27.780,154.718
C06211=1082.159,370.060,-97.652,176.485,27.774,154.717
C06212=1082.152,369.813,-97.615,176.482,27.768,154.715
C06213=1082.147,369.566,-97.578,176.479,27.761,154.714
C06214=1082.140,369.319,-97.541,176.475,27.755,154.713
C06215=1082.135,369.071,-97.504,176.472,27.749,154.712
C06216=1082.128,368.824,-97.468,176.468,27.743,154.711
C06217=1082.122,368.577,-97.430,176.465,27.737,154.710
C06218=1082.116,368.330,-97.394,176.461,27.731,154.709
C06219=1082.110,368.083,-97.357,176.458,27.725,154.708
C06220=1082.104,367.836,-97.320,176.454,27.719,154.707
C06221=1082.098,367.589,-97.284,176.452,27.712,154.705
C06222=1082.091,367.341,-97.247,176.448,27.706,154.704
C06223=1082.085,367.094,-97.210,176.445,27.700,154.703
C06224=1082.079,366.847,-97.173,176.441,27.694,154.702
C06225=1082.073,366.600,-97.137,176.438,27.688,154.701
C06226=1082.067,366.352,-97.100,176.434,27.682,154.700
C06227=1082.061,366.105,-97.063,176.431,27.676,154.699
C06228=1082.055,365.858,-97.026,176.428,27.670,154.698
C06229=1082.049,365.611,-96.990,176.425,27.664,154.697
C06230=1082.042,365.364,-96.953,176.422,27.658,154.696
C06231=1082.036,365.117,-96.917,176.418,27.652,154.695
C06232=1082.030,364.869,-96.881,176.415,27.647,154.694
C06233=1082.024,364.622,-96.844,176.411,27.641,154.693
C06234=1082.018,364.375,-96.808,176.408,27.635,154.691
C06235=1082.012,364.128,-96.771,176.404,27.629,154.690
C06236=1082.005,363.881,-96.735,176.401,27.623,154.689
C06237=1081.999,363.633,-96.699,176.397,27.617,154.688
C06238=1081.993,363.386,-96.663,176.395,27.611,154.687
C06239=1081.987,363.139,-96.626,176.391,27.605,154.686
C06240=1081.981,362.891,-96.590,176.388,27.600,154.685
C06241=1081.975,362.644,-96.554,176.385,27.594,154.684
C06242=1081.969,362.397,-96.517,176.381,27.588,154.683
C06243=1081.963,362.149,-96.481,176.378,27.582,154.682
C06244=1081.956,361.902,-96.445,176.374,27.576,154.681
C06245=1081.951,361.656,-96.409,176.371,27.571,154.680
C06246=1081.945,361.408,-96.373,176.367,27.565,154.679
C06247=1081.938,361.161,-96.337,176.364,27.559,154.678
C06248=1081.932,360.913,-96.301,176.361,27.554,154.677
C06249=1081.926,360.666,-96.264,176.358,27.548,154.676
C06250=1081.920,360.418,-96.229,176.355,27.542,154.675
C06251=1081.913,360.171,-96.192,176.351,27.537,154.674
C06252=1081.907,359.924,-96.157,176.348,27.531,154.673
C06253=1081.901,359.677,-96.120,176.345,27.525,154.672
C06254=1081.896,359.430,-96.085,176.341,27.519,154.671
C06255=1081.890,359.182,-96.049,176.338,27.514,154.670
C06256=1081.883,358.935,-96.013,176.335,27.508,154.669
C06257=1081.877,358.687,-95.977,176.331,27.503,154.668
C06258=1081.871,358.440,-95.941,176.328,27.497,154.667
C06259=1081.861,358.029,-95.882,176.322,27.488,154.665
C06260=1081.850,357.618,-95.822,176.317,27.479,154.664
C06261=1081.840,357.208,-95.763,176.312,27.470,154.662
C06262=1081.830,356.796,-95.704,176.306,27.461,154.661
C06263=1081.824,356.549,-95.667,176.303,27.455,154.660
C06264=1081.818,356.301,-95.632,176.300,27.449,154.659
C06265=1081.812,356.054,-95.597,176.297,27.444,154.658
C06266=1081.805,355.806,-95.561,176.293,27.438,154.657
C06267=1081.799,355.559,-95.525,176.290,27.432,154.656
C06268=1081.794,355.312,-95.490,176.287,27.427,154.655
C06269=1081.788,355.064,-95.454,176.283,27.422,154.654
C06270=1081.781,354.817,-95.419,176.280,27.416,154.653
C06271=1081.776,354.570,-95.384,176.277,27.411,154.652
C06272=1081.770,354.322,-95.348,176.273,27.405,154.651
C06273=1081.764,354.074,-95.312,176.270,27.400,154.650
C06274=1081.758,353.827,-95.276,176.267,27.394,154.649
C06275=1081.752,353.580,-95.242,176.263,27.389,154.648
C06276=1081.746,353.332,-95.206,176.260,27.384,154.647
C06277=1081.739,353.085,-95.170,176.257,27.378,154.646
C06278=1081.733,352.838,-95.135,176.253,27.373,154.646
C06279=1081.727,352.590,-95.100,176.251,27.367,154.645
C06280=1081.721,352.343,-95.064,176.248,27.362,154.644
C06281=1081.715,352.096,-95.029,176.245,27.357,154.643
C06282=1081.709,351.848,-94.993,176.241,27.351,154.642
C06283=1081.703,351.600,-94.959,176.238,27.346,154.641
C06284=1081.697,351.353,-94.924,176.235,27.341,154.640
C06285=1081.691,351.106,-94.888,176.231,27.335,154.639
C06286=1081.684,350.858,-94.853,176.228,27.330,154.638
C06287=1081.679,350.611,-94.818,176.225,27.325,154.637
C06288=1081.672,350.363,-94.783,176.222,27.320,154.636
C06289=1081.666,350.116,-94.747,176.218,27.315,154.636
C06290=1081.660,349.869,-94.712,176.215,27.309,154.635
C06291=1081.655,349.621,-94.677,176.212,27.304,154.634
C06292=1081.648,349.373,-94.642,176.208,27.299,154.633
C06293=1081.642,349.126,-94.607,176.205,27.293,154.632
C06294=1081.636,348.878,-94.573,176.202,27.288,154.631
C06295=1081.630,348.632,-94.537,176.199,27.283,154.630
C06296=1081.624,348.384,-94.503,176.195,27.278,154.629
C06297=1081.619,348.137,-94.467,176.192,27.273,154.628
C06298=1081.612,347.889,-94.433,176.189,27.267,154.628
C06299=1081.606,347.641,-94.397,176.186,27.262,154.627
C06300=1081.600,347.394,-94.363,176.182,27.257,154.626
C06301=1081.594,347.146,-94.327,176.179,27.252,154.625
C06302=1081.588,346.899,-94.293,176.176,27.247,154.624
C06303=1081.582,346.651,-94.258,176.173,27.242,154.623
C06304=1081.576,346.404,-94.224,176.170,27.237,154.622
C06305=1081.570,346.156,-94.188,176.166,27.231,154.621
C06306=1081.565,345.909,-94.154,176.163,27.226,154.621
C06307=1081.558,345.661,-94.119,176.160,27.221,154.620
C06308=1081.552,345.414,-94.085,176.157,27.216,154.619
C06309=1081.546,345.166,-94.050,176.153,27.211,154.618
C06310=1081.540,344.919,-94.016,176.151,27.206,154.617
C06311=1081.531,344.511,-93.958,176.145,27.197,154.616
C06312=1081.520,344.102,-93.901,176.140,27.189,154.614
C06313=1081.510,343.695,-93.844,176.135,27.181,154.613
C06314=1081.501,343.287,-93.787,176.130,27.173,154.612
C06315=1081.495,343.040,-93.753,176.126,27.168,154.611
C06316=1081.488,342.792,-93.718,176.123,27.163,154.610
C06317=1081.483,342.544,-93.684,176.120,27.158,154.609
C06318=1081.476,342.296,-93.650,176.117,27.153,154.608
C06319=1081.470,342.049,-93.616,176.114,27.148,154.608
C06320=1081.464,341.801,-93.581,176.110,27.143,154.607
C06321=1081.458,341.554,-93.546,176.107,27.138,154.606
C06322=1081.452,341.307,-93.512,176.104,27.133,154.605
C06323=1081.446,341.059,-93.478,176.101,27.128,154.604
C06324=1081.440,340.811,-93.443,176.098,27.123,154.603
C06325=1081.434,340.564,-93.409,176.095,27.118,154.603
C06326=1081.429,340.316,-93.374,176.091,27.113,154.602
C06327=1081.423,340.069,-93.340,176.088,27.108,154.601
C06328=1081.416,339.821,-93.306,176.085,27.103,154.600
C06329=1081.411,339.573,-93.273,176.082,27.098,154.599
C06330=1081.405,339.325,-93.239,176.079,27.094,154.599
C06331=1081.398,339.077,-93.204,176.076,27.088,154.598
C06332=1081.392,338.830,-93.170,176.073,27.084,154.597
C06333=1081.387,338.583,-93.136,176.070,27.079,154.596
C06334=1081.381,338.336,-93.102,176.066,27.074,154.595
C06335=1081.375,338.087,-93.067,176.063,27.069,154.595
C06336=1081.368,337.840,-93.034,176.060,27.064,154.594
C06337=1081.363,337.592,-93.000,176.057,27.060,154.593
C06338=1081.356,337.344,-92.966,176.054,27.055,154.592
C06339=1081.351,337.097,-92.932,176.051,27.050,154.592
C06340=1081.345,336.850,-92.898,176.048,27.045,154.591
C06341=1081.339,336.601,-92.864,176.045,27.041,154.590
C06342=1081.333,336.354,-92.830,176.041,27.035,154.589
C06343=1081.327,336.107,-92.796,176.038,27.031,154.588
C06344=1081.321,335.859,-92.763,176.035,27.026,154.588
C06345=1081.315,335.611,-92.728,176.032,27.021,154.587
C06346=1081.309,335.364,-92.694,176.029,27.016,154.586
C06347=1081.303,335.116,-92.661,176.026,27.012,154.585
C06348=1081.297,334.869,-92.627,176.023,27.007,154.585
C06349=1081.291,334.620,-92.594,176.020,27.003,154.584
C06350=1081.285,334.373,-92.559,176.017,26.998,154.583
C06351=1081.279,334.125,-92.525,176.014,26.993,154.582
C06352=1081.273,333.878,-92.492,176.011,26.988,154.582
C06353=1081.267,333.630,-92.458,176.007,26.983,154.581
C06354=1081.261,333.382,-92.424,176.004,26.978,154.580
C06355=1081.255,333.135,-92.391,176.001,26.974,154.579
C06356=1081.249,332.887,-92.358,175.998,26.969,154.579
C06357=1081.244,332.639,-92.324,175.995,26.964,154.578
C06358=1081.238,332.392,-92.290,175.992,26.960,154.577
C06359=1081.232,332.144,-92.257,175.989,26.955,154.576
C06360=1081.226,331.896,-92.222,175.986,26.951,154.576
C06361=1081.219,331.648,-92.190,175.983,26.946,154.575
C06362=1081.214,331.400,-92.156,175.980,26.941,154.574
C06363=1081.203,330.987,-92.100,175.974,26.933,154.573
C06364=1081.193,330.574,-92.044,175.969,26.926,154.572
C06365=1081.183,330.161,-91.989,175.964,26.919,154.570
C06366=1081.174,329.746,-91.933,175.959,26.911,154.569
C06367=1081.167,329.499,-91.900,175.956,26.906,154.568
C06368=1081.161,329.251,-91.867,175.953,26.902,154.568
C06369=1081.155,329.003,-91.834,175.950,26.897,154.567
C06370=1081.149,328.755,-91.800,175.947,26.893,154.566
C06371=1081.143,328.508,-91.767,175.943,26.888,154.566
C06372=1081.137,328.260,-91.733,175.940,26.884,154.565
C06373=1081.131,328.013,-91.701,175.937,26.879,154.564
C06374=1081.124,327.765,-91.668,175.934,26.875,154.564
C06375=1081.119,327.517,-91.635,175.931,26.870,154.563
C06376=1081.112,327.270,-91.602,175.928,26.866,154.562
C06377=1081.107,327.022,-91.569,175.925,26.861,154.561
C06378=1081.101,326.774,-91.536,175.922,26.857,154.561
C06379=1081.095,326.526,-91.502,175.919,26.852,154.560
C06380=1081.089,326.279,-91.470,175.916,26.848,154.559
C06381=1081.083,326.031,-91.436,175.913,26.844,154.559
C06382=1081.076,325.782,-91.403,175.910,26.839,154.558
C06383=1081.071,325.535,-91.370,175.907,26.834,154.557
C06384=1081.064,325.287,-91.337,175.904,26.830,154.556
C06385=1081.058,325.039,-91.304,175.901,26.825,154.556
C06386=1081.053,324.791,-91.271,175.898,26.821,154.555
C06387=1081.047,324.545,-91.239,175.895,26.817,154.555
C06388=1081.041,324.297,-91.205,175.892,26.812,154.554
C06389=1081.035,324.048,-91.173,175.888,26.808,154.553
C06390=1081.029,323.801,-91.141,175.885,26.803,154.552
C06391=1081.024,323.553,-91.107,175.882,26.799,154.552
C06392=1081.017,323.305,-91.075,175.879,26.794,154.551
C06393=1081.012,323.057,-91.041,175.876,26.790,154.550
C06394=1081.005,322.810,-91.008,175.873,26.785,154.550
C06395=1080.999,322.562,-90.976,175.870,26.781,154.549
C06396=1080.994,322.314,-90.943,175.867,26.776,154.548
C06397=1080.988,322.066,-90.910,175.864,26.772,154.548
C06398=1080.981,321.819,-90.878,175.861,26.767,154.547
C06399=1080.976,321.570,-90.845,175.858,26.763,154.546
C06400=1080.970,321.323,-90.813,175.855,26.759,154.546
C06401=1080.964,321.076,-90.780,175.852,26.754,154.545
C06402=1080.959,320.827,-90.747,175.850,26.750,154.544
C06403=1080.953,320.579,-90.714,175.847,26.746,154.543
C06404=1080.946,320.332,-90.682,175.844,26.741,154.543
C06405=1080.941,320.083,-90.649,175.840,26.737,154.542
C06406=1080.935,319.836,-90.617,175.837,26.733,154.542
C06407=1080.929,319.588,-90.585,175.834,26.728,154.541
C06408=1080.924,319.340,-90.551,175.831,26.724,154.540
C06409=1080.917,319.093,-90.519,175.828,26.719,154.539
C06410=1080.911,318.845,-90.487,175.825,26.715,154.539
C06411=1080.906,318.597,-90.454,175.822,26.711,154.538
C06412=1080.901,318.349,-90.422,175.819,26.706,154.537
C06413=1080.894,318.102,-90.389,175.816,26.702,154.537
C06414=1080.888,317.853,-90.357,175.814,26.697,154.536
C06415=1080.884,317.643,-90.330,175.811,26.694,154.536
C06416=1080.878,317.433,-90.302,175.808,26.690,154.535
C06417=1080.874,317.224,-90.275,175.806,26.687,154.534
C06418=1080.869,317.013,-90.247,175.803,26.683,154.534
C06419=1080.865,316.803,-90.219,175.801,26.679,154.533
C06420=1080.859,316.593,-90.192,175.799,26.675,154.533
C06421=1080.855,316.383,-90.165,175.795,26.672,154.532
C06422=1080.850,316.174,-90.137,175.793,26.668,154.532
C06423=1080.844,315.925,-90.105,175.790,26.664,154.531
C06424=1080.838,315.677,-90.073,175.787,26.659,154.530
C06425=1080.832,315.430,-90.041,175.785,26.655,154.530
C06426=1080.826,315.182,-90.009,175.782,26.651,154.529
C06427=1080.821,314.933,-89.976,175.779,26.646,154.528
C06428=1080.816,314.687,-89.944,175.776,26.642,154.528
C06429=1080.810,314.438,-89.911,175.773,26.638,154.527
C06430=1080.803,314.190,-89.880,175.770,26.634,154.526
C06431=1080.797,313.942,-89.848,175.767,26.629,154.526
C06432=1080.791,313.694,-89.816,175.763,26.626,154.525
C06433=1080.785,313.447,-89.784,175.761,26.622,154.525
C06434=1080.779,313.199,-89.752,175.758,26.617,154.524
C06435=1080.773,312.951,-89.720,175.755,26.613,154.523
C06436=1080.767,312.704,-89.689,175.752,26.609,154.523
C06437=1080.761,312.455,-89.656,175.749,26.605,154.522
C06438=1080.755,312.207,-89.624,175.746,26.600,154.521
C06439=1080.749,311.959,-89.592,175.743,26.597,154.521
C06440=1080.743,311.712,-89.561,175.740,26.592,154.520
C06441=1080.737,311.464,-89.529,175.737,26.588,154.520
C06442=1080.731,311.216,-89.497,175.734,26.584,154.519
C06443=1080.725,310.968,-89.465,175.731,26.580,154.518
C06444=1080.719,310.720,-89.433,175.728,26.576,154.518
C06445=1080.713,310.473,-89.402,175.725,26.571,154.517
C06446=1080.707,310.225,-89.370,175.722,26.568,154.517
C06447=1080.701,309.977,-89.338,175.720,26.564,154.516
C06448=1080.695,309.729,-89.307,175.717,26.559,154.515
C06449=1080.689,309.480,-89.275,175.714,26.555,154.515
C06450=1080.683,309.232,-89.243,175.711,26.551,154.514
C06451=1080.678,308.985,-89.212,175.707,26.547,154.513
C06452=1080.671,308.737,-89.180,175.704,26.543,154.513
C06453=1080.666,308.489,-89.149,175.701,26.539,154.512
C06454=1080.660,308.241,-89.117,175.699,26.535,154.512
C06455=1080.654,307.994,-89.086,175.696,26.531,154.511
C06456=1080.648,307.746,-89.054,175.693,26.526,154.510
C06457=1080.643,307.498,-89.023,175.690,26.523,154.510
C06458=1080.637,307.249,-88.991,175.687,26.518,154.509
C06459=1080.631,307.002,-88.959,175.685,26.514,154.509
C06460=1080.625,306.754,-88.927,175.681,26.510,154.508
C06461=1080.619,306.506,-88.896,175.678,26.506,154.507
C06462=1080.613,306.258,-88.865,175.675,26.502,154.507
C06463=1080.607,306.010,-88.833,175.672,26.498,154.506
C06464=1080.601,305.763,-88.802,175.669,26.493,154.506
C06465=1080.595,305.515,-88.770,175.667,26.490,154.505
C06466=1080.590,305.266,-88.739,175.664,26.486,154.504
C06467=1080.584,305.019,-88.708,175.661,26.481,154.504
C06468=1080.578,304.771,-88.676,175.658,26.477,154.503
C06469=1080.573,304.523,-88.645,175.655,26.473,154.503
C06470=1080.566,304.275,-88.614,175.652,26.470,154.502
C06471=1080.557,303.858,-88.561,175.647,26.462,154.501
C06472=1080.547,303.441,-88.508,175.642,26.456,154.500
C06473=1080.538,303.024,-88.455,175.637,26.449,154.499
C06474=1080.527,302.607,-88.403,175.633,26.442,154.498
C06475=1080.522,302.358,-88.372,175.629,26.438,154.497
C06476=1080.515,302.111,-88.341,175.627,26.434,154.497
C06477=1080.510,301.863,-88.310,175.624,26.430,154.496
C06478=1080.504,301.615,-88.278,175.621,26.426,154.496
C06479=1080.499,301.367,-88.248,175.618,26.421,154.495
C06480=1080.493,301.119,-88.217,175.615,26.417,154.494
C06481=1080.487,300.871,-88.185,175.613,26.413,154.494
C06482=1080.482,300.623,-88.154,175.610,26.410,154.493
C06483=1080.475,300.376,-88.123,175.607,26.405,154.493
C06484=1080.470,300.128,-88.092,175.603,26.401,154.492
C06485=1080.464,299.879,-88.062,175.601,26.397,154.491
C06486=1080.459,299.632,-88.030,175.598,26.393,154.491
C06487=1080.453,299.384,-88.000,175.595,26.389,154.490
C06488=1080.448,299.136,-87.969,175.592,26.385,154.490
C06489=1080.441,298.888,-87.937,175.590,26.381,154.489
C06490=1080.436,298.640,-87.906,175.587,26.377,154.489
C06491=1080.431,298.391,-87.875,175.584,26.373,154.488
C06492=1080.425,298.144,-87.845,175.581,26.369,154.487
C06493=1080.418,297.896,-87.813,175.579,26.365,154.487
C06494=1080.413,297.648,-87.783,175.575,26.361,154.486
C06495=1080.407,297.400,-87.752,175.572,26.357,154.486
C06496=1080.401,297.151,-87.721,175.570,26.353,154.485
C06497=1080.396,296.903,-87.691,175.567,26.349,154.485
C06498=1080.390,296.656,-87.659,175.564,26.345,154.484
C06499=1080.384,296.408,-87.629,175.561,26.341,154.483
C06500=1080.378,296.160,-87.598,175.559,26.338,154.483
C06501=1080.372,295.911,-87.567,175.556,26.333,154.482
C06502=1080.367,295.664,-87.537,175.553,26.329,154.482
C06503=1080.361,295.416,-87.507,175.549,26.326,154.481
C06504=1080.354,295.167,-87.476,175.547,26.322,154.481
C06505=1080.349,294.919,-87.446,175.544,26.318,154.480
C06506=1080.344,294.671,-87.415,175.541,26.314,154.479
C06507=1080.338,294.424,-87.384,175.539,26.310,154.479
C06508=1080.332,294.176,-87.354,175.536,26.306,154.478
C06509=1080.325,293.927,-87.323,175.533,26.302,154.478
C06510=1080.320,293.679,-87.293,175.530,26.298,154.477
C06511=1080.314,293.432,-87.263,175.527,26.295,154.477
C06512=1080.309,293.183,-87.232,175.524,26.291,154.476
C06513=1080.303,292.936,-87.201,175.521,26.286,154.476
C06514=1080.297,292.687,-87.171,175.519,26.283,154.475
C06515=1080.291,292.439,-87.140,175.516,26.279,154.474
C06516=1080.285,292.191,-87.110,175.513,26.275,154.474
C06517=1080.279,291.944,-87.080,175.510,26.272,154.473
C06518=1080.274,291.695,-87.050,175.507,26.267,154.473
C06519=1080.268,291.447,-87.020,175.504,26.263,154.472
C06520=1080.261,291.199,-86.989,175.502,26.260,154.472
C06521=1080.255,290.951,-86.958,175.499,26.256,154.471
C06522=1080.250,290.703,-86.928,175.496,26.252,154.471
C06523=1080.241,290.300,-86.879,175.491,26.245,154.470
C06524=1080.232,289.898,-86.830,175.487,26.239,154.469
C06525=1080.222,289.494,-86.781,175.482,26.233,154.468
C06526=1080.212,289.092,-86.732,175.478,26.227,154.467
C06527=1080.207,288.844,-86.702,175.475,26.223,154.467
C06528=1080.201,288.596,-86.672,175.472,26.219,154.466
C06529=1080.195,288.348,-86.641,175.469,26.215,154.466
C06530=1080.189,288.100,-86.612,175.467,26.212,154.465
C06531=1080.183,287.851,-86.582,175.464,26.208,154.464
C06532=1080.177,287.603,-86.552,175.461,26.204,154.464
C06533=1080.171,287.355,-86.522,175.459,26.200,154.463
C06534=1080.166,287.107,-86.491,175.455,26.197,154.463
C06535=1080.160,286.859,-86.462,175.453,26.193,154.462
C06536=1080.154,286.611,-86.431,175.450,26.189,154.462
C06537=1080.148,286.363,-86.402,175.447,26.185,154.461
C06538=1080.142,286.115,-86.372,175.445,26.181,154.461
C06539=1080.137,285.867,-86.342,175.442,26.177,154.460
C06540=1080.131,285.619,-86.312,175.439,26.173,154.460
C06541=1080.125,285.370,-86.282,175.436,26.170,154.459
C06542=1080.119,285.122,-86.252,175.433,26.166,154.459
C06543=1080.113,284.874,-86.223,175.430,26.162,154.458
C06544=1080.107,284.627,-86.193,175.428,26.159,154.458
C06545=1080.102,284.378,-86.163,175.425,26.155,154.457
C06546=1080.096,284.130,-86.133,175.423,26.151,154.456
C06547=1080.091,283.882,-86.103,175.420,26.147,154.456
C06548=1080.084,283.634,-86.074,175.417,26.143,154.455
C06549=1080.079,283.385,-86.044,175.414,26.140,154.455
C06550=1080.073,283.137,-86.014,175.411,26.136,154.454
C06551=1080.067,282.889,-85.984,175.408,26.132,154.454
C06552=1080.061,282.641,-85.955,175.406,26.128,154.453
C06553=1080.055,282.393,-85.925,175.403,26.124,154.453
C06554=1080.050,282.145,-85.895,175.401,26.120,154.452
C06555=1080.044,281.896,-85.866,175.398,26.117,154.452
C06556=1080.038,281.648,-85.837,175.395,26.113,154.451
C06557=1080.032,281.400,-85.806,175.392,26.109,154.451
C06558=1080.027,281.152,-85.777,175.389,26.105,154.450
C06559=1080.022,280.904,-85.747,175.387,26.102,154.450
C06560=1080.016,280.656,-85.718,175.384,26.098,154.449
C06561=1080.010,280.407,-85.689,175.381,26.094,154.449
C06562=1080.004,280.160,-85.659,175.379,26.090,154.448
C06563=1079.998,279.911,-85.629,175.376,26.086,154.447
C06564=1079.993,279.663,-85.600,175.373,26.083,154.447
C06565=1079.986,279.415,-85.571,175.370,26.079,154.447
C06566=1079.981,279.166,-85.541,175.368,26.076,154.446
C06567=1079.975,278.918,-85.512,175.365,26.072,154.446
C06568=1079.969,278.670,-85.482,175.362,26.068,154.445
C06569=1079.963,278.422,-85.453,175.360,26.064,154.444
C06570=1079.957,278.173,-85.424,175.357,26.061,154.444
C06571=1079.952,277.926,-85.394,175.354,26.057,154.443
C06572=1079.946,277.677,-85.365,175.351,26.053,154.443
C06573=1079.941,277.429,-85.336,175.348,26.049,154.442
C06574=1079.934,277.181,-85.307,175.346,26.046,154.442
C06575=1079.925,276.788,-85.260,175.341,26.040,154.441
C06576=1079.916,276.395,-85.214,175.338,26.034,154.440
C06577=1079.908,276.002,-85.168,175.333,26.028,154.439
C06578=1079.898,275.610,-85.121,175.328,26.022,154.439
C06579=1079.892,275.361,-85.092,175.326,26.018,154.438
C06580=1079.886,275.113,-85.064,175.323,26.015,154.438
C06581=1079.881,274.864,-85.034,175.321,26.011,154.437
C06582=1079.874,274.616,-85.005,175.318,26.007,154.437
C06583=1079.869,274.368,-84.976,175.316,26.004,154.436
C06584=1079.863,274.120,-84.947,175.312,26.000,154.436
C06585=1079.857,273.872,-84.918,175.309,25.996,154.435
C06586=1079.852,273.623,-84.889,175.307,25.993,154.435
C06587=1079.846,273.375,-84.860,175.304,25.989,154.434
C06588=1079.841,273.127,-84.830,175.302,25.985,154.434
C06589=1079.835,272.878,-84.802,175.299,25.981,154.433
C06590=1079.828,272.630,-84.773,175.297,25.978,154.433
C06591=1079.822,272.382,-84.744,175.293,25.974,154.432
C06592=1079.817,272.134,-84.715,175.291,25.971,154.432
C06593=1079.811,271.886,-84.686,175.288,25.967,154.431
C06594=1079.805,271.638,-84.657,175.286,25.963,154.430
C06595=1079.800,271.389,-84.628,175.283,25.959,154.430
C06596=1079.794,271.141,-84.600,175.281,25.956,154.430
C06597=1079.788,270.893,-84.571,175.278,25.952,154.429
C06598=1079.782,270.644,-84.542,175.275,25.948,154.429
C06599=1079.777,270.396,-84.513,175.272,25.945,154.428
C06600=1079.771,270.148,-84.484,175.269,25.941,154.428
C06601=1079.765,269.900,-84.456,175.267,25.937,154.427
C06602=1079.759,269.651,-84.427,175.264,25.934,154.427
C06603=1079.754,269.403,-84.398,175.262,25.930,154.426
C06604=1079.748,269.155,-84.369,175.259,25.926,154.426
C06605=1079.742,268.906,-84.341,175.256,25.923,154.425
C06606=1079.736,268.658,-84.312,175.253,25.919,154.425
C06607=1079.730,268.410,-84.284,175.251,25.916,154.424
C06608=1079.724,268.162,-84.255,175.248,25.912,154.424
C06609=1079.719,267.913,-84.226,175.246,25.908,154.423
C06610=1079.714,267.665,-84.198,175.243,25.904,154.423
C06611=1079.707,267.417,-84.169,175.241,25.901,154.422
C06612=1079.701,267.168,-84.140,175.237,25.897,154.422
C06613=1079.696,266.920,-84.112,175.235,25.894,154.421
C06614=1079.690,266.672,-84.083,175.232,25.890,154.421
C06615=1079.684,266.424,-84.055,175.230,25.887,154.420
C06616=1079.678,266.176,-84.026,175.227,25.883,154.420
C06617=1079.672,265.927,-83.998,175.225,25.879,154.419
C06618=1079.668,265.678,-83.970,175.222,25.875,154.419
C06619=1079.661,265.430,-83.940,175.219,25.872,154.418
C06620=1079.655,265.182,-83.912,175.216,25.868,154.418
C06621=1079.650,264.933,-83.884,175.214,25.865,154.417
C06622=1079.644,264.685,-83.855,175.211,25.861,154.417
C06623=1079.638,264.437,-83.827,175.209,25.857,154.416
C06624=1079.633,264.189,-83.799,175.206,25.854,154.416
C06625=1079.627,263.941,-83.771,175.204,25.850,154.415
C06626=1079.621,263.692,-83.743,175.201,25.847,154.415
C06627=1079.612,263.302,-83.699,175.197,25.841,154.414
C06628=1079.602,262.912,-83.654,175.193,25.836,154.413
C06629=1079.593,262.522,-83.609,175.188,25.830,154.413
C06630=1079.584,262.133,-83.565,175.185,25.824,154.412
C06631=1079.578,261.884,-83.537,175.181,25.821,154.411
C06632=1079.572,261.635,-83.509,175.179,25.817,154.411
C06633=1079.566,261.387,-83.481,175.176,25.814,154.410
C06634=1079.560,261.139,-83.453,175.174,25.810,154.410
C06635=1079.555,260.891,-83.425,175.171,25.806,154.409
C06636=1079.549,260.642,-83.397,175.169,25.803,154.409
C06637=1079.543,260.394,-83.369,175.166,25.799,154.408
C06638=1079.537,260.145,-83.341,175.163,25.796,154.408
C06639=1079.531,259.897,-83.313,175.161,25.792,154.407
C06640=1079.525,259.649,-83.285,175.158,25.789,154.407
C06641=1079.519,259.400,-83.257,175.156,25.785,154.407
C06642=1079.513,259.152,-83.229,175.153,25.781,154.406
C06643=1079.507,258.903,-83.201,175.151,25.778,154.406
C06644=1079.502,258.655,-83.173,175.147,25.774,154.405
C06645=1079.495,258.407,-83.145,175.145,25.771,154.405
C06646=1079.490,258.159,-83.117,175.142,25.767,154.404
C06647=1079.484,257.910,-83.089,175.140,25.764,154.404
C06648=1079.479,257.662,-83.061,175.138,25.760,154.403
C06649=1079.472,257.413,-83.034,175.135,25.756,154.403
C06650=1079.467,257.165,-83.006,175.132,25.753,154.402
C06651=1079.461,256.916,-82.978,175.129,25.749,154.402
C06652=1079.455,256.668,-82.950,175.127,25.746,154.401
C06653=1079.450,256.420,-82.922,175.124,25.742,154.401
C06654=1079.444,256.171,-82.895,175.122,25.739,154.400
C06655=1079.439,255.923,-82.867,175.120,25.735,154.400
C06656=1079.432,255.675,-82.839,175.117,25.732,154.399
C06657=1079.427,255.426,-82.811,175.114,25.728,154.399
C06658=1079.421,255.177,-82.783,175.111,25.725,154.398
C06659=1079.415,254.929,-82.756,175.109,25.721,154.398
C06660=1079.410,254.681,-82.728,175.107,25.717,154.397
C06661=1079.404,254.433,-82.700,175.104,25.714,154.397
C06662=1079.398,254.184,-82.673,175.102,25.710,154.397
C06663=1079.393,253.936,-82.645,175.099,25.706,154.396
C06664=1079.386,253.688,-82.617,175.096,25.703,154.396
C06665=1079.381,253.439,-82.590,175.093,25.699,154.395
C06666=1079.375,253.190,-82.562,175.091,25.696,154.395
C06667=1079.370,252.969,-82.538,175.089,25.693,154.394
C06668=1079.365,252.749,-82.513,175.087,25.689,154.394
C06669=1079.360,252.527,-82.488,175.084,25.686,154.393
C06670=1079.354,252.307,-82.464,175.082,25.683,154.393
C06671=1079.350,252.086,-82.440,175.080,25.680,154.392
C06672=1079.345,251.865,-82.416,175.078,25.677,154.392
C06673=1079.339,251.644,-82.390,175.076,25.673,154.392
C06674=1079.335,251.422,-82.366,175.073,25.670,154.391
C06675=1079.329,251.175,-82.339,175.071,25.667,154.391
C06676=1079.323,250.925,-82.311,175.068,25.663,154.390
C06677=1079.317,250.678,-82.284,175.066,25.660,154.390
C06678=1079.312,250.429,-82.257,175.063,25.656,154.389
C06679=1079.307,250.205,-82.232,175.061,25.653,154.389
C06680=1079.301,249.981,-82.207,175.058,25.649,154.388
C06681=1079.297,249.758,-82.182,175.056,25.646,154.388
C06682=1079.291,249.535,-82.158,175.054,25.643,154.387
C06683=1079.287,249.310,-82.133,175.052,25.640,154.387
C06684=1079.281,249.087,-82.109,175.050,25.636,154.387
C06685=1079.277,248.863,-82.084,175.047,25.633,154.386
C06686=1079.271,248.639,-82.059,175.045,25.630,154.386
C06687=1079.266,248.391,-82.032,175.043,25.626,154.385
C06688=1079.261,248.142,-82.005,175.040,25.622,154.385
C06689=1079.255,247.894,-81.977,175.038,25.619,154.384
C06690=1079.249,247.645,-81.950,175.035,25.616,154.384
C06691=1079.243,247.396,-81.923,175.032,25.612,154.383
C06692=1079.238,247.148,-81.895,175.030,25.608,154.383
C06693=1079.232,246.900,-81.868,175.028,25.605,154.382
C06694=1079.226,246.651,-81.841,175.025,25.601,154.382
C06695=1079.221,246.402,-81.814,175.023,25.598,154.381
C06696=1079.215,246.155,-81.787,175.020,25.594,154.381
C06697=1079.209,245.906,-81.760,175.018,25.590,154.380
C06698=1079.204,245.658,-81.733,175.015,25.587,154.380
C06699=1079.197,245.408,-81.706,175.012,25.583,154.379
C06700=1079.192,245.160,-81.679,175.010,25.579,154.379
C06701=1079.186,244.912,-81.651,175.008,25.576,154.379
C06702=1079.180,244.664,-81.625,175.005,25.572,154.378
C06703=1079.175,244.415,-81.597,175.003,25.569,154.378
C06704=1079.169,244.166,-81.570,175.001,25.566,154.377
C06705=1079.163,243.918,-81.544,174.997,25.562,154.377
C06706=1079.158,243.669,-81.516,174.995,25.559,154.376
C06707=1079.152,243.421,-81.490,174.993,25.555,154.376
C06708=1079.146,243.173,-81.462,174.990,25.551,154.375
C06709=1079.141,242.924,-81.436,174.988,25.548,154.375
C06710=1079.136,242.676,-81.409,174.986,25.544,154.374
C06711=1079.129,242.427,-81.382,174.983,25.540,154.374
C06712=1079.123,242.178,-81.355,174.980,25.537,154.373
C06713=1079.118,241.930,-81.328,174.978,25.534,154.373
C06714=1079.112,241.682,-81.302,174.975,25.530,154.372
C06715=1079.106,241.433,-81.275,174.973,25.526,154.372
C06716=1079.100,241.185,-81.248,174.971,25.523,154.371
C06717=1079.095,240.936,-81.221,174.968,25.519,154.371
C06718=1079.089,240.687,-81.194,174.966,25.516,154.371
C06719=1079.083,240.439,-81.167,174.963,25.513,154.370
C06720=1079.078,240.190,-81.141,174.960,25.509,154.370
C06721=1079.072,239.941,-81.115,174.958,25.506,154.369
C06722=1079.066,239.693,-81.088,174.956,25.502,154.369
C06723=1079.060,239.445,-81.062,174.953,25.498,154.368
C06724=1079.055,239.196,-81.035,174.951,25.495,154.368
C06725=1079.049,238.948,-81.008,174.949,25.492,154.367
C06726=1079.042,238.699,-80.981,174.946,25.488,154.367
C06727=1079.037,238.451,-80.955,174.943,25.484,154.366
C06728=1079.031,238.202,-80.929,174.941,25.481,154.366
C06729=1079.025,237.953,-80.902,174.939,25.477,154.365
C06730=1079.020,237.705,-80.875,174.936,25.474,154.365
C06731=1079.014,237.457,-80.849,174.934,25.470,154.364
C06732=1079.008,237.208,-80.823,174.932,25.467,154.364
C06733=1079.003,236.959,-80.796,174.929,25.463,154.363
C06734=1078.997,236.711,-80.769,174.926,25.459,154.363
C06735=1078.988,236.312,-80.727,174.923,25.454,154.362
C06736=1078.979,235.911,-80.684,174.919,25.449,154.362
C06737=1078.969,235.513,-80.642,174.915,25.442,154.361
C06738=1078.961,235.113,-80.600,174.911,25.437,154.360
C06739=1078.955,234.865,-80.573,174.909,25.433,154.359
C06740=1078.949,234.616,-80.546,174.907,25.430,154.359
C06741=1078.944,234.367,-80.520,174.904,25.426,154.359
C06742=1078.938,234.119,-80.494,174.901,25.423,154.358
C06743=1078.932,233.871,-80.467,174.899,25.420,154.358
C06744=1078.926,233.622,-80.442,174.896,25.416,154.357
C06745=1078.920,233.374,-80.415,174.894,25.412,154.357
C06746=1078.915,233.125,-80.389,174.892,25.409,154.356
C06747=1078.909,232.876,-80.362,174.890,25.405,154.356
C06748=1078.904,232.627,-80.337,174.887,25.402,154.355
C06749=1078.898,232.379,-80.310,174.885,25.398,154.355
C06750=1078.892,232.130,-80.284,174.882,25.395,154.354
C06751=1078.886,231.882,-80.258,174.880,25.391,154.354
C06752=1078.880,231.633,-80.232,174.877,25.387,154.353
C06753=1078.875,231.385,-80.205,174.875,25.384,154.353
C06754=1078.869,231.136,-80.179,174.873,25.380,154.352
C06755=1078.864,230.888,-80.153,174.871,25.377,154.352
C06756=1078.859,230.639,-80.127,174.868,25.373,154.352
C06757=1078.852,230.390,-80.102,174.866,25.370,154.351
C06758=1078.847,230.142,-80.075,174.863,25.367,154.351
C06759=1078.841,229.893,-80.049,174.861,25.363,154.350
C06760=1078.835,229.645,-80.023,174.858,25.359,154.350
C06761=1078.829,229.396,-79.997,174.856,25.356,154.349
C06762=1078.824,229.147,-79.971,174.854,25.353,154.349
C06763=1078.817,228.899,-79.945,174.852,25.349,154.348
C06764=1078.812,228.650,-79.919,174.849,25.346,154.348
C06765=1078.806,228.401,-79.893,174.846,25.342,154.347
C06766=1078.800,228.153,-79.867,174.844,25.338,154.347
C06767=1078.795,227.905,-79.842,174.842,25.335,154.346
C06768=1078.789,227.656,-79.816,174.839,25.331,154.346
C06769=1078.783,227.407,-79.791,174.837,25.328,154.345
C06770=1078.777,227.159,-79.764,174.835,25.324,154.345
C06771=1078.771,226.910,-79.739,174.833,25.321,154.345
C06772=1078.766,226.661,-79.713,174.830,25.317,154.344
C06773=1078.760,226.412,-79.687,174.827,25.314,154.344
C06774=1078.754,226.165,-79.661,174.825,25.310,154.343
C06775=1078.749,225.916,-79.635,174.823,25.307,154.343
C06776=1078.743,225.667,-79.610,174.821,25.304,154.342
C06777=1078.737,225.418,-79.584,174.818,25.300,154.342
C06778=1078.732,225.169,-79.558,174.816,25.296,154.341
C06779=1078.726,224.920,-79.533,174.814,25.293,154.341
C06780=1078.721,224.672,-79.507,174.811,25.290,154.340
C06781=1078.714,224.424,-79.481,174.809,25.286,154.340
C06782=1078.709,224.175,-79.455,174.806,25.282,154.339
C06783=1078.702,223.926,-79.430,174.804,25.279,154.339
C06784=1078.698,223.678,-79.404,174.802,25.275,154.338
C06785=1078.692,223.429,-79.378,174.800,25.272,154.338
C06786=1078.686,223.180,-79.353,174.797,25.268,154.338
C06787=1078.677,222.773,-79.311,174.793,25.262,154.337
C06788=1078.668,222.365,-79.269,174.790,25.257,154.336
C06789=1078.659,221.957,-79.227,174.786,25.251,154.335
C06790=1078.648,221.549,-79.185,174.783,25.245,154.334
C06791=1078.643,221.301,-79.160,174.780,25.241,154.334
C06792=1078.637,221.052,-79.134,174.777,25.238,154.334
C06793=1078.631,220.804,-79.109,174.775,25.234,154.333
C06794=1078.626,220.555,-79.083,174.773,25.231,154.333
C06795=1078.620,220.306,-79.059,174.771,25.228,154.332
C06796=1078.614,220.057,-79.033,174.768,25.224,154.332
C06797=1078.609,219.808,-79.007,174.766,25.221,154.331
C06798=1078.602,219.560,-78.982,174.764,25.217,154.331
C06799=1078.597,219.312,-78.957,174.761,25.214,154.330
C06800=1078.591,219.063,-78.931,174.759,25.210,154.330
C06801=1078.585,218.814,-78.906,174.757,25.207,154.329
C06802=1078.580,218.566,-78.882,174.754,25.203,154.329
C06803=1078.574,218.317,-78.856,174.752,25.200,154.328
C06804=1078.568,218.068,-78.830,174.750,25.196,154.328
C06805=1078.563,217.820,-78.805,174.748,25.193,154.328
C06806=1078.557,217.571,-78.779,174.746,25.189,154.327
C06807=1078.551,217.322,-78.755,174.743,25.185,154.326
C06808=1078.546,217.074,-78.730,174.740,25.182,154.326
C06809=1078.539,216.825,-78.704,174.738,25.178,154.326
C06810=1078.534,216.575,-78.679,174.736,25.175,154.325
C06811=1078.529,216.327,-78.654,174.734,25.172,154.325
C06812=1078.522,216.079,-78.629,174.732,25.168,154.324
C06813=1078.516,215.830,-78.604,174.730,25.165,154.324
C06814=1078.512,215.581,-78.579,174.727,25.161,154.323
C06815=1078.505,215.333,-78.553,174.725,25.158,154.323
C06816=1078.500,215.085,-78.528,174.723,25.154,154.322
C06817=1078.494,214.835,-78.504,174.721,25.150,154.322
C06818=1078.488,214.586,-78.478,174.718,25.147,154.321
C06819=1078.483,214.338,-78.454,174.716,25.143,154.321
C06820=1078.477,214.089,-78.428,174.713,25.140,154.320
C06821=1078.471,213.841,-78.403,174.711,25.136,154.320
C06822=1078.466,213.592,-78.378,174.709,25.133,154.319
C06823=1078.461,213.344,-78.353,174.707,25.129,154.319
C06824=1078.455,213.094,-78.328,174.705,25.126,154.318
C06825=1078.448,212.846,-78.303,174.703,25.122,154.318
C06826=1078.443,212.597,-78.279,174.700,25.119,154.318
C06827=1078.437,212.348,-78.254,174.697,25.115,154.317
C06828=1078.432,212.100,-78.229,174.695,25.112,154.317
C06829=1078.426,211.851,-78.203,174.693,25.108,154.316
C06830=1078.421,211.602,-78.179,174.691,25.104,154.316
C06831=1078.415,211.354,-78.154,174.689,25.101,154.315
C06832=1078.409,211.104,-78.129,174.687,25.097,154.315
C06833=1078.403,210.856,-78.104,174.685,25.094,154.314
C06834=1078.397,210.607,-78.080,174.683,25.091,154.314
C06835=1078.392,210.358,-78.055,174.680,25.087,154.313
C06836=1078.386,210.110,-78.030,174.677,25.083,154.313
C06837=1078.381,209.861,-78.006,174.675,25.080,154.312
C06838=1078.374,209.612,-77.980,174.673,25.077,154.312
C06839=1078.365,209.209,-77.941,174.670,25.071,154.311
C06840=1078.356,208.805,-77.901,174.666,25.065,154.310
C06841=1078.347,208.402,-77.861,174.663,25.059,154.310
C06842=1078.337,207.998,-77.821,174.659,25.054,154.309
C06843=1078.314,206.962,-77.720,174.552,24.997,154.310
C06844=1078.308,206.713,-77.697,174.549,24.994,154.310
C06845=1078.303,206.465,-77.673,174.547,24.991,154.309
C06846=1078.298,206.216,-77.648,174.545,24.989,154.309
C06847=1078.292,205.967,-77.624,174.542,24.987,154.309
C06848=1078.286,205.719,-77.600,174.540,24.984,154.309
C06849=1078.281,205.469,-77.577,174.538,24.981,154.308
C06850=1078.275,205.221,-77.552,174.535,24.979,154.308
C06851=1078.269,204.972,-77.528,174.533,24.976,154.308
C06852=1078.263,204.723,-77.504,174.530,24.974,154.308
C06853=1078.258,204.475,-77.480,174.528,24.971,154.307
C06854=1078.252,204.226,-77.457,174.526,24.969,154.307
C06855=1078.247,203.977,-77.433,174.523,24.966,154.307
C06856=1078.241,203.728,-77.408,174.521,24.963,154.307
C06857=1078.235,203.479,-77.385,174.519,24.961,154.306
C06858=1078.230,203.230,-77.361,174.516,24.958,154.306
C06859=1078.225,202.982,-77.337,174.514,24.956,154.306
C06860=1078.219,202.733,-77.314,174.513,24.954,154.306
C06861=1078.214,202.484,-77.289,174.510,24.951,154.305
C06862=1078.207,202.235,-77.265,174.508,24.948,154.305
C06863=1078.202,201.986,-77.242,174.506,24.946,154.305
C06864=1078.196,201.738,-77.218,174.503,24.944,154.305
C06865=1078.190,201.489,-77.195,174.501,24.941,154.304
C06866=1078.184,201.240,-77.171,174.498,24.938,154.304
C06867=1078.178,200.991,-77.147,174.496,24.936,154.304
C06868=1078.173,200.742,-77.123,174.494,24.934,154.304
C06869=1078.167,200.494,-77.100,174.491,24.931,154.304
C06870=1078.162,200.245,-77.076,174.489,24.928,154.303
C06871=1078.156,199.996,-77.052,174.487,24.926,154.303
C06872=1078.150,199.747,-77.029,174.484,24.923,154.303
C06873=1078.145,199.498,-77.005,174.482,24.921,154.303
C06874=1078.139,199.249,-76.982,174.479,24.919,154.302
C06875=1078.133,199.001,-76.958,174.477,24.916,154.302
C06876=1078.128,198.752,-76.935,174.475,24.913,154.302
C06877=1078.122,198.504,-76.911,174.472,24.911,154.302
C06878=1078.116,198.254,-76.887,174.470,24.909,154.301
C06879=1078.110,198.005,-76.864,174.468,24.906,154.301
C06880=1078.105,197.757,-76.841,174.465,24.903,154.301
C06881=1078.099,197.508,-76.816,174.464,24.901,154.301
C06882=1078.094,197.259,-76.793,174.461,24.899,154.301
C06883=1078.088,197.010,-76.770,174.459,24.896,154.300
C06884=1078.083,196.762,-76.746,174.457,24.894,154.300
C06885=1078.077,196.513,-76.723,174.455,24.891,154.300
C06886=1078.071,196.264,-76.700,174.452,24.889,154.300
C06887=1078.065,196.014,-76.676,174.450,24.886,154.299
C06888=1078.059,195.766,-76.653,174.447,24.884,154.299
C06889=1078.053,195.517,-76.629,174.445,24.881,154.299
C06890=1078.048,195.268,-76.606,174.443,24.879,154.299
C06891=1078.043,195.019,-76.583,174.440,24.876,154.298
C06892=1078.037,194.770,-76.560,174.438,24.873,154.298
C06893=1078.032,194.522,-76.535,174.437,24.871,154.298
C06894=1078.026,194.273,-76.512,174.434,24.869,154.298
C06895=1078.020,194.024,-76.489,174.432,24.866,154.297
C06896=1078.015,193.775,-76.465,174.429,24.864,154.297
C06897=1078.009,193.526,-76.442,174.427,24.861,154.297
C06898=1078.003,193.278,-76.419,174.425,24.859,154.297
C06899=1077.998,193.029,-76.396,174.422,24.856,154.296
C06900=1077.992,192.780,-76.372,174.420,24.854,154.296
C06901=1077.987,192.531,-76.349,174.418,24.851,154.296
C06902=1077.981,192.282,-76.326,174.416,24.849,154.296
C06903=1077.976,192.033,-76.303,174.414,24.846,154.295
C06904=1077.969,191.753,-76.277,174.411,24.843,154.295
C06905=1077.962,191.473,-76.250,174.408,24.840,154.295
C06906=1077.957,191.192,-76.225,174.406,24.838,154.295
C06907=1077.951,190.912,-76.199,174.404,24.835,154.294
C06908=1077.945,190.663,-76.176,174.401,24.832,154.294
C06909=1077.940,190.414,-76.152,174.399,24.830,154.294
C06910=1077.934,190.165,-76.129,174.397,24.828,154.294
C06911=1077.928,189.917,-76.106,174.394,24.825,154.293
C06912=1077.922,189.668,-76.083,174.392,24.822,154.293
C06913=1077.917,189.419,-76.059,174.390,24.820,154.293
C06914=1077.912,189.170,-76.036,174.388,24.818,154.293
C06915=1077.906,188.921,-76.013,174.386,24.815,154.292
C06916=1077.901,188.673,-75.991,174.384,24.812,154.292
C06917=1077.896,188.424,-75.967,174.381,24.810,154.292
C06918=1077.890,188.175,-75.944,174.379,24.807,154.292
C06919=1077.884,187.926,-75.921,174.376,24.805,154.291
C06920=1077.879,187.677,-75.898,174.375,24.803,154.291
C06921=1077.873,187.428,-75.875,174.373,24.800,154.291
C06922=1077.868,187.179,-75.852,174.370,24.797,154.291
C06923=1077.862,186.930,-75.829,174.368,24.795,154.290
C06924=1077.857,186.682,-75.806,174.366,24.792,154.290
C06925=1077.851,186.433,-75.783,174.363,24.790,154.290
C06926=1077.846,186.184,-75.760,174.362,24.788,154.290
C06927=1077.841,185.935,-75.737,174.360,24.785,154.289
C06928=1077.835,185.685,-75.715,174.357,24.782,154.289
C06929=1077.829,185.436,-75.692,174.355,24.780,154.289
C06930=1077.824,185.188,-75.669,174.353,24.777,154.289
C06931=1077.819,184.939,-75.646,174.350,24.775,154.288
C06932=1077.813,184.691,-75.623,174.349,24.772,154.288
C06933=1077.807,184.442,-75.600,174.347,24.770,154.288
C06934=1077.801,184.193,-75.577,174.344,24.768,154.288
C06935=1077.795,183.944,-75.556,174.342,24.765,154.288
C06936=1077.789,183.695,-75.533,174.339,24.763,154.287
C06937=1077.784,183.446,-75.510,174.337,24.760,154.287
C06938=1077.778,183.197,-75.487,174.336,24.758,154.287
C06939=1077.772,182.948,-75.464,174.333,24.756,154.287
C06940=1077.766,182.699,-75.442,174.331,24.753,154.286
C06941=1077.760,182.450,-75.419,174.328,24.751,154.286
C06942=1077.755,182.202,-75.397,174.326,24.748,154.286
C06943=1077.749,181.953,-75.374,174.325,24.746,154.286
C06944=1077.743,181.704,-75.352,174.322,24.744,154.286
C06945=1077.738,181.455,-75.329,174.320,24.741,154.285
C06946=1077.732,181.206,-75.306,174.318,24.739,154.285
C06947=1077.726,180.956,-75.284,174.315,24.736,154.285
C06948=1077.721,180.707,-75.261,174.314,24.734,154.285
C06949=1077.714,180.459,-75.239,174.311,24.732,154.284
C06950=1077.709,180.210,-75.217,174.309,24.729,154.284
C06951=1077.704,179.961,-75.194,174.307,24.727,154.284
C06952=1077.697,179.712,-75.172,174.305,24.725,154.284
C06953=1077.692,179.463,-75.149,174.303,24.722,154.283
C06954=1077.686,179.214,-75.126,174.301,24.719,154.283
C06955=1077.680,178.965,-75.103,174.298,24.717,154.283
C06956=1077.675,178.717,-75.082,174.296,24.715,154.283
C06957=1077.669,178.468,-75.059,174.294,24.712,154.283
C06958=1077.664,178.218,-75.037,174.292,24.710,154.282
C06959=1077.658,177.969,-75.014,174.290,24.708,154.282
C06960=1077.651,177.721,-74.992,174.287,24.705,154.282
C06961=1077.647,177.472,-74.970,174.286,24.703,154.282
C06962=1077.641,177.223,-74.947,174.283,24.700,154.281
C06963=1077.635,176.974,-74.925,174.281,24.698,154.281
C06964=1077.629,176.725,-74.902,174.279,24.696,154.281
C06965=1077.624,176.476,-74.880,174.276,24.693,154.281
C06966=1077.618,176.228,-74.858,174.275,24.691,154.280
C06967=1077.612,175.978,-74.836,174.273,24.688,154.280
C06968=1077.606,175.697,-74.810,174.270,24.686,154.280
C06969=1077.600,175.417,-74.785,174.268,24.683,154.280
C06970=1077.594,175.136,-74.760,174.266,24.680,154.280
C06971=1077.586,174.856,-74.735,174.263,24.678,154.279
C06972=1077.581,174.607,-74.713,174.261,24.675,154.279
C06973=1077.576,174.358,-74.691,174.259,24.672,154.279
C06974=1077.570,174.109,-74.669,174.256,24.670,154.278
C06975=1077.564,173.860,-74.646,174.255,24.668,154.278
C06976=1077.559,173.611,-74.624,174.253,24.665,154.278
C06977=1077.553,173.362,-74.602,174.250,24.663,154.278
C06978=1077.547,173.113,-74.580,174.248,24.660,154.278
C06979=1077.542,172.864,-74.557,174.246,24.658,154.277
C06980=1077.536,172.615,-74.536,174.244,24.655,154.277
C06981=1077.531,172.366,-74.514,174.242,24.653,154.277
C06982=1077.525,172.118,-74.492,174.240,24.651,154.277
C06983=1077.519,171.868,-74.469,174.238,24.648,154.276
C06984=1077.514,171.619,-74.447,174.236,24.646,154.276
C06985=1077.508,171.371,-74.425,174.233,24.643,154.276
C06986=1077.503,171.121,-74.403,174.232,24.641,154.276
C06987=1077.497,170.872,-74.381,174.230,24.639,154.275
C06988=1077.492,170.623,-74.359,174.227,24.636,154.275
C06989=1077.486,170.375,-74.336,174.226,24.634,154.275
C06990=1077.480,170.126,-74.315,174.223,24.631,154.275
C06991=1077.475,169.876,-74.293,174.221,24.629,154.274
C06992=1077.469,169.627,-74.271,174.219,24.626,154.274
C06993=1077.464,169.379,-74.249,174.217,24.624,154.274
C06994=1077.458,169.130,-74.227,174.215,24.622,154.274
C06995=1077.453,168.881,-74.205,174.213,24.619,154.274
C06996=1077.447,168.632,-74.183,174.211,24.617,154.273
C06997=1077.441,168.382,-74.161,174.209,24.614,154.273
C06998=1077.436,168.134,-74.139,174.207,24.611,154.273
C06999=1077.430,167.885,-74.117,174.205,24.609,154.273
C07000=1077.425,167.636,-74.095,174.203,24.607,154.272
C07001=1077.420,167.387,-74.073,174.201,24.604,154.272
C07002=1077.414,167.138,-74.052,174.198,24.601,154.272
C07003=1077.409,166.889,-74.030,174.197,24.599,154.271
C07004=1077.403,166.640,-74.008,174.194,24.597,154.271
C07005=1077.398,166.391,-73.986,174.192,24.594,154.271
C07006=1077.392,166.143,-73.964,174.191,24.592,154.271
C07007=1077.386,165.893,-73.942,174.188,24.589,154.270
C07008=1077.381,165.645,-73.921,174.186,24.587,154.270
C07009=1077.375,165.395,-73.898,174.185,24.585,154.270
C07010=1077.370,165.147,-73.877,174.182,24.582,154.270
C07011=1077.364,164.897,-73.855,174.180,24.579,154.270
C07012=1077.359,164.649,-73.834,174.179,24.577,154.269
C07013=1077.353,164.399,-73.811,174.176,24.574,154.269
C07014=1077.349,164.150,-73.789,174.174,24.572,154.269
C07015=1077.342,163.901,-73.768,174.173,24.570,154.269
C07016=1077.338,163.652,-73.746,174.170,24.567,154.268
C07017=1077.331,163.403,-73.724,174.168,24.565,154.268
C07018=1077.327,163.154,-73.702,174.167,24.562,154.268
C07019=1077.320,162.905,-73.681,174.164,24.560,154.267
C07020=1077.316,162.656,-73.659,174.162,24.557,154.267
C07021=1077.309,162.407,-73.637,174.161,24.555,154.267
C07022=1077.304,162.159,-73.616,174.158,24.552,154.267
C07023=1077.299,161.910,-73.594,174.156,24.550,154.266
C07024=1077.293,161.660,-73.573,174.154,24.547,154.266
C07025=1077.288,161.411,-73.551,174.152,24.545,154.266
C07026=1077.282,161.162,-73.530,174.150,24.542,154.266
C07027=1077.277,160.913,-73.509,174.149,24.540,154.265
C07028=1077.271,160.664,-73.486,174.146,24.538,154.265
C07029=1077.266,160.415,-73.465,174.145,24.535,154.265
C07030=1077.260,160.166,-73.443,174.142,24.532,154.265
C07031=1077.254,159.917,-73.423,174.140,24.530,154.265
C07032=1077.248,159.636,-73.398,174.138,24.528,154.264
C07033=1077.241,159.355,-73.374,174.136,24.524,154.264
C07034=1077.235,159.074,-73.350,174.133,24.522,154.264
C07035=1077.229,158.793,-73.326,174.131,24.519,154.263
C07036=1077.223,158.544,-73.304,174.129,24.517,154.263
C07037=1077.217,158.295,-73.283,174.127,24.515,154.263
C07038=1077.212,158.046,-73.262,174.126,24.512,154.263
C07039=1077.206,157.797,-73.241,174.123,24.510,154.262
C07040=1077.200,157.548,-73.219,174.121,24.507,154.262
C07041=1077.195,157.299,-73.197,174.120,24.505,154.262
C07042=1077.189,157.050,-73.176,174.117,24.502,154.262
C07043=1077.184,156.801,-73.155,174.115,24.500,154.261
C07044=1077.178,156.552,-73.134,174.114,24.497,154.261
C07045=1077.172,156.303,-73.112,174.111,24.495,154.261
C07046=1077.166,156.054,-73.091,174.110,24.493,154.261
C07047=1077.161,155.805,-73.070,174.108,24.490,154.260
C07048=1077.156,155.556,-73.048,174.105,24.487,154.260
C07049=1077.150,155.306,-73.027,174.104,24.486,154.260
C07050=1077.145,155.058,-73.006,174.101,24.483,154.260
C07051=1077.139,154.808,-72.985,174.100,24.481,154.259
C07052=1077.133,154.560,-72.964,174.098,24.478,154.259
C07053=1077.128,154.311,-72.943,174.095,24.476,154.259
C07054=1077.122,154.061,-72.922,174.094,24.473,154.259
C07055=1077.116,153.813,-72.900,174.092,24.471,154.259
C07056=1077.110,153.563,-72.879,174.090,24.468,154.258
C07057=1077.105,153.315,-72.858,174.088,24.466,154.258
C07058=1077.099,153.066,-72.837,174.086,24.464,154.258
C07059=1077.093,152.816,-72.816,174.084,24.461,154.258
C07060=1077.088,152.568,-72.795,174.082,24.459,154.257
C07061=1077.082,152.319,-72.774,174.080,24.457,154.257
C07062=1077.076,152.069,-72.753,174.078,24.454,154.257
C07063=1077.071,151.820,-72.732,174.076,24.451,154.257
C07064=1077.065,151.571,-72.710,174.074,24.449,154.256
C07065=1077.060,151.322,-72.690,174.072,24.446,154.256
C07066=1077.054,151.073,-72.669,174.071,24.445,154.256
C07067=1077.048,150.824,-72.648,174.068,24.442,154.256
C07068=1077.043,150.575,-72.626,174.067,24.440,154.255
C07069=1077.037,150.326,-72.606,174.065,24.437,154.255
C07070=1077.032,150.077,-72.585,174.062,24.435,154.255
C07071=1077.026,149.828,-72.564,174.061,24.432,154.255
C07072=1077.021,149.578,-72.543,174.059,24.430,154.254
C07073=1077.015,149.330,-72.522,174.057,24.427,154.254
C07074=1077.009,149.080,-72.501,174.055,24.425,154.254
C07075=1077.003,148.832,-72.480,174.053,24.423,154.254
C07076=1076.998,148.583,-72.460,174.051,24.420,154.253
C07077=1076.992,148.333,-72.439,174.049,24.417,154.253
C07078=1076.986,148.085,-72.417,174.048,24.415,154.253
C07079=1076.981,147.835,-72.397,174.045,24.412,154.253
C07080=1076.975,147.586,-72.376,174.044,24.411,154.252
C07081=1076.969,147.337,-72.355,174.041,24.408,154.252
C07082=1076.964,147.088,-72.335,174.040,24.406,154.252
C07083=1076.958,146.839,-72.314,174.038,24.403,154.252
C07084=1076.952,146.590,-72.293,174.035,24.401,154.251
C07085=1076.947,146.341,-72.272,174.034,24.398,154.251
C07086=1076.941,146.092,-72.252,174.032,24.396,154.251
C07087=1076.935,145.842,-72.231,174.030,24.393,154.251
C07088=1076.930,145.594,-72.210,174.028,24.391,154.250
C07089=1076.924,145.345,-72.189,174.027,24.389,154.250
C07090=1076.918,145.096,-72.169,174.024,24.386,154.250
C07091=1076.912,144.846,-72.148,174.023,24.384,154.250
C07092=1076.907,144.597,-72.127,174.021,24.381,154.249
C07093=1076.902,144.348,-72.107,174.019,24.379,154.249
C07094=1076.896,144.099,-72.087,174.017,24.377,154.249
C07095=1076.890,143.850,-72.066,174.015,24.374,154.249
C07096=1076.884,143.569,-72.043,174.013,24.372,154.248
C07097=1076.877,143.288,-72.019,174.011,24.369,154.248
C07098=1076.871,143.007,-71.996,174.009,24.366,154.248
C07099=1076.864,142.725,-71.972,174.006,24.363,154.247
C07100=1076.859,142.476,-71.952,174.005,24.361,154.247
C07101=1076.853,142.227,-71.932,174.003,24.358,154.247
C07102=1076.848,141.978,-71.911,174.000,24.356,154.247
C07103=1076.843,141.729,-71.891,173.999,24.353,154.246
C07104=1076.836,141.480,-71.870,173.997,24.351,154.246
C07105=1076.831,141.231,-71.849,173.995,24.348,154.246
C07106=1076.825,140.982,-71.828,173.993,24.346,154.246
C07107=1076.819,140.733,-71.808,173.992,24.344,154.246
C07108=1076.814,140.484,-71.788,173.989,24.341,154.245
C07109=1076.809,140.235,-71.767,173.988,24.339,154.245
C07110=1076.802,139.985,-71.747,173.986,24.336,154.245
C07111=1076.797,139.736,-71.726,173.984,24.334,154.244
C07112=1076.792,139.487,-71.706,173.982,24.332,154.244
C07113=1076.786,139.238,-71.686,173.980,24.329,154.244
C07114=1076.780,138.989,-71.665,173.978,24.326,154.244
C07115=1076.774,138.740,-71.645,173.977,24.324,154.243
C07116=1076.769,138.490,-71.625,173.975,24.321,154.243
C07117=1076.763,138.241,-71.605,173.973,24.319,154.243
C07118=1076.757,137.992,-71.584,173.971,24.317,154.243
C07119=1076.752,137.743,-71.563,173.969,24.315,154.242
C07120=1076.746,137.494,-71.543,173.967,24.312,154.242
C07121=1076.741,137.245,-71.523,173.966,24.310,154.242
C07122=1076.734,136.996,-71.503,173.964,24.307,154.242
C07123=1076.729,136.747,-71.482,173.962,24.305,154.241
C07124=1076.723,136.498,-71.462,173.960,24.302,154.241
C07125=1076.718,136.249,-71.442,173.958,24.300,154.241
C07126=1076.712,136.000,-71.422,173.956,24.297,154.241
C07127=1076.707,135.750,-71.402,173.955,24.295,154.240
C07128=1076.701,135.501,-71.382,173.952,24.292,154.240
C07129=1076.696,135.252,-71.361,173.951,24.290,154.240
C07130=1076.690,135.003,-71.341,173.949,24.288,154.240
C07131=1076.683,134.754,-71.321,173.947,24.285,154.239
C07132=1076.678,134.505,-71.300,173.945,24.283,154.239
C07133=1076.672,134.256,-71.280,173.944,24.280,154.239
C07134=1076.667,134.006,-71.261,173.941,24.278,154.239
C07135=1076.661,133.757,-71.241,173.940,24.275,154.238
C07136=1076.655,133.508,-71.220,173.938,24.273,154.238
C07137=1076.649,133.259,-71.200,173.936,24.271,154.238
C07138=1076.644,133.010,-71.180,173.935,24.268,154.238
C07139=1076.639,132.761,-71.160,173.933,24.266,154.237
C07140=1076.633,132.512,-71.140,173.931,24.263,154.237
C07141=1076.627,132.263,-71.120,173.929,24.261,154.237
C07142=1076.622,132.014,-71.099,173.928,24.258,154.236
C07143=1076.616,131.764,-71.080,173.925,24.256,154.236
C07144=1076.610,131.515,-71.060,173.924,24.254,154.236
C07145=1076.604,131.266,-71.040,173.922,24.251,154.236
C07146=1076.598,131.017,-71.020,173.920,24.249,154.235
C07147=1076.593,130.767,-71.000,173.918,24.246,154.235
C07148=1076.587,130.519,-70.980,173.916,24.244,154.235
C07149=1076.581,130.270,-70.960,173.914,24.241,154.235
C07150=1076.575,130.020,-70.941,173.913,24.239,154.234
C07151=1076.570,129.771,-70.920,173.911,24.236,154.234
C07152=1076.564,129.522,-70.900,173.909,24.234,154.234
C07153=1076.558,129.273,-70.881,173.908,24.232,154.234
C07154=1076.552,129.024,-70.861,173.905,24.229,154.234
C07155=1076.546,128.775,-70.841,173.904,24.227,154.233
C07156=1076.541,128.525,-70.821,173.902,24.224,154.233
C07157=1076.535,128.276,-70.801,173.900,24.222,154.233
C07158=1076.529,128.027,-70.782,173.898,24.219,154.232
C07159=1076.523,127.778,-70.762,173.897,24.218,154.232
C07160=1076.517,127.496,-70.739,173.895,24.214,154.232
C07161=1076.511,127.216,-70.717,173.892,24.212,154.232
C07162=1076.504,126.934,-70.695,173.891,24.209,154.231
C07163=1076.497,126.653,-70.673,173.889,24.207,154.231
C07164=1076.492,126.403,-70.653,173.886,24.204,154.231
C07165=1076.486,126.154,-70.633,173.885,24.201,154.231
C07166=1076.480,125.905,-70.613,173.883,24.199,154.230
C07167=1076.474,125.656,-70.594,173.881,24.196,154.230
C07168=1076.469,125.407,-70.574,173.880,24.194,154.230
C07169=1076.463,125.158,-70.554,173.878,24.191,154.229
C07170=1076.458,124.908,-70.534,173.876,24.189,154.229
C07171=1076.452,124.659,-70.515,173.874,24.187,154.229
C07172=1076.446,124.410,-70.495,173.873,24.184,154.229
C07173=1076.440,124.161,-70.475,173.870,24.182,154.228
C07174=1076.434,123.912,-70.456,173.869,24.179,154.228
C07175=1076.428,123.663,-70.436,173.868,24.177,154.228
C07176=1076.423,123.414,-70.417,173.865,24.174,154.228
C07177=1076.418,123.164,-70.397,173.864,24.172,154.227
C07178=1076.412,122.916,-70.377,173.862,24.169,154.227
C07179=1076.407,122.666,-70.358,173.860,24.167,154.227
C07180=1076.401,122.417,-70.338,173.858,24.165,154.227
C07181=1076.395,122.168,-70.319,173.857,24.162,154.226
C07182=1076.389,121.918,-70.300,173.855,24.160,154.226
C07183=1076.383,121.670,-70.280,173.853,24.157,154.226
C07184=1076.378,121.420,-70.261,173.852,24.155,154.225
C07185=1076.372,121.171,-70.240,173.849,24.152,154.225
C07186=1076.367,120.922,-70.221,173.848,24.150,154.225
C07187=1076.362,120.673,-70.202,173.847,24.147,154.225
C07188=1076.356,120.424,-70.182,173.845,24.145,154.224
C07189=1076.350,120.175,-70.163,173.843,24.142,154.224
C07190=1076.344,119.925,-70.143,173.841,24.140,154.224
C07191=1076.338,119.676,-70.124,173.840,24.137,154.224
C07192=1076.332,119.427,-70.104,173.838,24.135,154.223
C07193=1076.327,119.178,-70.085,173.836,24.132,154.223
C07194=1076.321,118.928,-70.066,173.835,24.130,154.223
C07195=1076.316,118.680,-70.046,173.832,24.127,154.222
C07196=1076.310,118.431,-70.027,173.831,24.125,154.222
C07197=1076.305,118.181,-70.007,173.829,24.122,154.222
C07198=1076.299,117.931,-69.988,173.827,24.120,154.222
C07199=1076.293,117.683,-69.968,173.826,24.117,154.221
C07200=1076.288,117.434,-69.949,173.824,24.115,154.221
C07201=1076.283,117.184,-69.930,173.822,24.112,154.221
C07202=1076.277,116.935,-69.910,173.821,24.110,154.220
C07203=1076.271,116.686,-69.891,173.819,24.107,154.220
C07204=1076.265,116.437,-69.871,173.817,24.105,154.220
C07205=1076.260,116.188,-69.852,173.815,24.102,154.220
C07206=1076.254,115.939,-69.833,173.814,24.100,154.219
C07207=1076.249,115.689,-69.814,173.813,24.097,154.219
C07208=1076.243,115.440,-69.795,173.810,24.095,154.219
C07209=1076.237,115.190,-69.775,173.809,24.092,154.219
C07210=1076.232,114.942,-69.757,173.807,24.090,154.218
C07211=1076.226,114.693,-69.737,173.805,24.087,154.218
C07212=1076.221,114.443,-69.717,173.804,24.085,154.218
C07213=1076.215,114.194,-69.698,173.802,24.082,154.217
C07214=1076.209,113.944,-69.679,173.800,24.080,154.217
C07215=1076.204,113.696,-69.660,173.798,24.077,154.217
C07216=1076.198,113.446,-69.641,173.797,24.075,154.217
C07217=1076.192,113.197,-69.622,173.795,24.072,154.216
C07218=1076.186,112.948,-69.603,173.793,24.070,154.216
C07219=1076.181,112.698,-69.584,173.792,24.067,154.216
C07220=1076.176,112.450,-69.565,173.790,24.065,154.215
C07221=1076.170,112.200,-69.545,173.788,24.062,154.215
C07222=1076.164,111.951,-69.526,173.787,24.060,154.215
C07223=1076.158,111.702,-69.508,173.785,24.057,154.215
C07224=1076.151,111.420,-69.486,173.783,24.054,154.214
C07225=1076.145,111.139,-69.464,173.781,24.051,154.214
C07226=1076.139,110.858,-69.442,173.779,24.049,154.214
C07227=1076.132,110.576,-69.421,173.778,24.046,154.213
C07228=1076.127,110.327,-69.403,173.775,24.044,154.213
C07229=1076.121,110.078,-69.384,173.774,24.041,154.213
C07230=1076.115,109.829,-69.365,173.773,24.039,154.213
C07231=1076.109,109.579,-69.346,173.770,24.036,154.212
C07232=1076.103,109.330,-69.327,173.769,24.034,154.212
C07233=1076.098,109.081,-69.308,173.768,24.031,154.212
C07234=1076.092,108.832,-69.289,173.765,24.029,154.212
C07235=1076.086,108.583,-69.270,173.764,24.026,154.211
C07236=1076.080,108.333,-69.251,173.763,24.024,154.211
C07237=1076.074,108.085,-69.233,173.761,24.021,154.211
C07238=1076.069,107.835,-69.213,173.759,24.019,154.210
C07239=1076.063,107.585,-69.195,173.757,24.016,154.210
C07240=1076.058,107.337,-69.176,173.756,24.014,154.210
C07241=1076.052,107.088,-69.157,173.754,24.011,154.210
C07242=1076.046,106.838,-69.138,173.752,24.009,154.209
C07243=1076.040,106.589,-69.119,173.751,24.006,154.209
C07244=1076.035,106.340,-69.100,173.749,24.004,154.209
C07245=1076.029,106.090,-69.082,173.747,24.001,154.208
C07246=1076.023,105.841,-69.063,173.746,23.999,154.208
C07247=1076.018,105.592,-69.044,173.744,23.996,154.208
C07248=1076.012,105.343,-69.025,173.742,23.994,154.208
C07249=1076.006,105.094,-69.006,173.741,23.991,154.207
C07250=1076.001,104.844,-68.988,173.739,23.989,154.207
C07251=1075.995,104.595,-68.969,173.737,23.986,154.207
C07252=1075.989,104.346,-68.950,173.736,23.984,154.206
C07253=1075.984,104.097,-68.932,173.735,23.982,154.206
C07254=1075.978,103.847,-68.914,173.732,23.978,154.206
C07255=1075.972,103.598,-68.894,173.731,23.976,154.206
C07256=1075.967,103.349,-68.876,173.730,23.974,154.205
C07257=1075.961,103.099,-68.858,173.728,23.971,154.205
